gfCNCPoint5[25189] = {X 489.1455, Y 22.6360, Z -7.1667, A 0.000, B 0.000, C 0.000 }
gfCNCPoint5[25190] = {X 493.1303, Y 22.2874, Z -7.1667, A 0.000, B 0.000, C 0.000 }
gfCNCPoint5[25191] = {X 485.1607, Y 22.3674, Z -7.1667, A 0.000, B 0.000, C 0.000 }
gfCNCPoint5[25192] = {X 489.1455, Y 22.7160, Z -7.1667, A 0.000, B 0.000, C 0.000 }
gfCNCPoint5[25193] = {X 493.5290, Y 22.7160, Z -7.1667, A 0.000, B 0.000, C 0.000 }
gfCNCPoint5[25194] = {X 493.5290, Y 19.6226, Z -7.1667, A 0.000, B 0.000, C 0.000 }
gfCNCPoint5[25195] = {X 487.6640, Y 19.6221, Z -7.1667, A 0.000, B 0.000, C 0.000 }
gfCNCPoint5[25196] = {X 486.9712, Y 19.6268, Z -7.1667, A 0.000, B 0.000, C 0.000 }
gfCNCPoint5[25197] = {X 485.8542, Y 19.6990, Z -7.1667, A 0.000, B 0.000, C 0.000 }
gfCNCPoint5[25198] = {X 484.7569, Y 19.9204, Z -7.1667, A 0.000, B 0.000, C 0.000 }
gfCNCPoint5[25199] = {X 484.5580, Y 20.0321, Z -7.1667, A 0.000, B 0.000, C 0.000 }
gfCNCPoint5[25200] = {X 484.4352, Y 20.2245, Z -7.1667, A 0.000, B 0.000, C 0.000 }
gfCNCPoint5[25201] = {X 484.2684, Y 20.9674, Z -7.1667, A 0.000, B 0.000, C 0.000 }
gfCNCPoint5[25202] = {X 484.2552, Y 21.7288, Z -7.1667, A 0.000, B 0.000, C 0.000 }
gfCNCPoint5[25203] = {X 484.3961, Y 22.4771, Z -7.1667, A 0.000, B 0.000, C 0.000 }
gfCNCPoint5[25204] = {X 484.6514, Y 22.5532, Z -7.1667, A 0.000, B 0.000, C 0.000 }
gfCNCPoint5[25205] = {X 484.9147, Y 22.5933, Z -7.1667, A 0.000, B 0.000, C 0.000 }
gfCNCPoint5[25206] = {X 486.2771, Y 22.6950, Z -7.1667, A 0.000, B 0.000, C 0.000 }
gfCNCPoint5[25207] = {X 487.6431, Y 22.7160, Z -7.1667, A 0.000, B 0.000, C 0.000 }
gfCNCPoint5[25208] = {X 489.1455, Y 22.7160, Z -7.1667, A 0.000, B 0.000, C 0.000 }
gfCNCPoint5[25209] = {X 493.1303, Y 22.3674, Z -7.1667, A 0.000, B 0.000, C 0.000 }
gfCNCPoint5[25210] = {X 485.1607, Y 22.4474, Z -7.1667, A 0.000, B 0.000, C 0.000 }
gfCNCPoint5[25211] = {X 489.1455, Y 22.7960, Z -7.1667, A 0.000, B 0.000, C 0.000 }
gfCNCPoint5[25212] = {X 493.6090, Y 22.7960, Z -7.1667, A 0.000, B 0.000, C 0.000 }
gfCNCPoint5[25213] = {X 493.6090, Y 19.5426, Z -7.1667, A 0.000, B 0.000, C 0.000 }
gfCNCPoint5[25214] = {X 487.6637, Y 19.5421, Z -7.1667, A 0.000, B 0.000, C 0.000 }
gfCNCPoint5[25215] = {X 486.9710, Y 19.5468, Z -7.1667, A 0.000, B 0.000, C 0.000 }
gfCNCPoint5[25216] = {X 485.8434, Y 19.6197, Z -7.1667, A 0.000, B 0.000, C 0.000 }
gfCNCPoint5[25217] = {X 484.7359, Y 19.8432, Z -7.1667, A 0.000, B 0.000, C 0.000 }
gfCNCPoint5[25218] = {X 484.5030, Y 19.9740, Z -7.1667, A 0.000, B 0.000, C 0.000 }
gfCNCPoint5[25219] = {X 484.3593, Y 20.1991, Z -7.1667, A 0.000, B 0.000, C 0.000 }
gfCNCPoint5[25220] = {X 484.1874, Y 20.9710, Z -7.1667, A 0.000, B 0.000, C 0.000 }
gfCNCPoint5[25221] = {X 484.1778, Y 21.7618, Z -7.1667, A 0.000, B 0.000, C 0.000 }
gfCNCPoint5[25222] = {X 484.3308, Y 22.5376, Z -7.1667, A 0.000, B 0.000, C 0.000 }
gfCNCPoint5[25223] = {X 484.6140, Y 22.6267, Z -7.1667, A 0.000, B 0.000, C 0.000 }
gfCNCPoint5[25224] = {X 484.9073, Y 22.6730, Z -7.1667, A 0.000, B 0.000, C 0.000 }
gfCNCPoint5[25225] = {X 486.2736, Y 22.7749, Z -7.1667, A 0.000, B 0.000, C 0.000 }
gfCNCPoint5[25226] = {X 487.6437, Y 22.7960, Z -7.1667, A 0.000, B 0.000, C 0.000 }
gfCNCPoint5[25227] = {X 489.1455, Y 22.7960, Z -7.1667, A 0.000, B 0.000, C 0.000 }
gfCNCPoint5[25228] = {X 493.1303, Y 22.4474, Z -7.1667, A 0.000, B 0.000, C 0.000 }
gfCNCPoint5[25229] = {X 485.1607, Y 22.5274, Z -7.1667, A 0.000, B 0.000, C 0.000 }
gfCNCPoint5[25230] = {X 489.1455, Y 22.8760, Z -7.1667, A 0.000, B 0.000, C 0.000 }
gfCNCPoint5[25231] = {X 493.6890, Y 22.8760, Z -7.1667, A 0.000, B 0.000, C 0.000 }
gfCNCPoint5[25232] = {X 493.6890, Y 19.4626, Z -7.1667, A 0.000, B 0.000, C 0.000 }
gfCNCPoint5[25233] = {X 487.6634, Y 19.4621, Z -7.1667, A 0.000, B 0.000, C 0.000 }
gfCNCPoint5[25234] = {X 486.9708, Y 19.4668, Z -7.1667, A 0.000, B 0.000, C 0.000 }
gfCNCPoint5[25235] = {X 485.8327, Y 19.5404, Z -7.1667, A 0.000, B 0.000, C 0.000 }
gfCNCPoint5[25236] = {X 484.7148, Y 19.7660, Z -7.1667, A 0.000, B 0.000, C 0.000 }
gfCNCPoint5[25237] = {X 484.4481, Y 19.9159, Z -7.1667, A 0.000, B 0.000, C 0.000 }
gfCNCPoint5[25238] = {X 484.2835, Y 20.1737, Z -7.1667, A 0.000, B 0.000, C 0.000 }
gfCNCPoint5[25239] = {X 484.1065, Y 20.9744, Z -7.1667, A 0.000, B 0.000, C 0.000 }
gfCNCPoint5[25240] = {X 484.1005, Y 21.7943, Z -7.1667, A 0.000, B 0.000, C 0.000 }
gfCNCPoint5[25241] = {X 484.2657, Y 22.5974, Z -7.1667, A 0.000, B 0.000, C 0.000 }
gfCNCPoint5[25242] = {X 484.5771, Y 22.7001, Z -7.1667, A 0.000, B 0.000, C 0.000 }
gfCNCPoint5[25243] = {X 484.9007, Y 22.7527, Z -7.1667, A 0.000, B 0.000, C 0.000 }
gfCNCPoint5[25244] = {X 486.2706, Y 22.8548, Z -7.1667, A 0.000, B 0.000, C 0.000 }
gfCNCPoint5[25245] = {X 487.6442, Y 22.8760, Z -7.1667, A 0.000, B 0.000, C 0.000 }
gfCNCPoint5[25246] = {X 489.1455, Y 22.8760, Z -7.1667, A 0.000, B 0.000, C 0.000 }
gfCNCPoint5[25247] = {X 493.1303, Y 22.5274, Z -7.1667, A 0.000, B 0.000, C 0.000 }
gfCNCPoint5[25248] = {X 489.1455, Y 20.9560, Z -7.1667, A 0.000, B 0.000, C 0.000 }
gfCNCPoint5[25249] = {X 489.1455, Y 22.9560, Z -7.1667, A 0.000, B 0.000, C 0.000 }
gfCNCPoint5[25250] = {X 493.7690, Y 22.9560, Z -7.1667, A 0.000, B 0.000, C 0.000 }
gfCNCPoint5[25251] = {X 493.7690, Y 19.3826, Z -7.1667, A 0.000, B 0.000, C 0.000 }
gfCNCPoint5[25252] = {X 487.6632, Y 19.3821, Z -7.1667, A 0.000, B 0.000, C 0.000 }
gfCNCPoint5[25253] = {X 486.9707, Y 19.3868, Z -7.1667, A 0.000, B 0.000, C 0.000 }
gfCNCPoint5[25254] = {X 485.8220, Y 19.4611, Z -7.1667, A 0.000, B 0.000, C 0.000 }
gfCNCPoint5[25255] = {X 484.6937, Y 19.6888, Z -7.1667, A 0.000, B 0.000, C 0.000 }
gfCNCPoint5[25256] = {X 484.3931, Y 19.8577, Z -7.1667, A 0.000, B 0.000, C 0.000 }
gfCNCPoint5[25257] = {X 484.2076, Y 20.1484, Z -7.1667, A 0.000, B 0.000, C 0.000 }
gfCNCPoint5[25258] = {X 484.0256, Y 20.9775, Z -7.1667, A 0.000, B 0.000, C 0.000 }
gfCNCPoint5[25259] = {X 484.0233, Y 21.8264, Z -7.1667, A 0.000, B 0.000, C 0.000 }
gfCNCPoint5[25260] = {X 484.2007, Y 22.6566, Z -7.1667, A 0.000, B 0.000, C 0.000 }
gfCNCPoint5[25261] = {X 484.5397, Y 22.7732, Z -7.1667, A 0.000, B 0.000, C 0.000 }
gfCNCPoint5[25262] = {X 484.8932, Y 22.8324, Z -7.1667, A 0.000, B 0.000, C 0.000 }
gfCNCPoint5[25263] = {X 486.2672, Y 22.9348, Z -7.1667, A 0.000, B 0.000, C 0.000 }
gfCNCPoint5[25264] = {X 487.6448, Y 22.9560, Z -7.1667, A 0.000, B 0.000, C 0.000 }
gfCNCPoint5[25265] = {X 489.1455, Y 22.9560, Z -7.1667, A 0.000, B 0.000, C 0.000 }
gfCNCPoint5[25266] = {X 493.1455, Y 22.9560, Z -7.1667, A 0.000, B 0.000, C 0.000 }
gfCNCPoint5[25267] = {X 493.1455, Y 22.9560, Z -4.1667, A 0.000, B 0.000, C 0.000 }
gfCNCPoint5[25268] = {X 493.1455, Y 22.9560, Z 11.0000, A 0.000, B 0.000, C 0.000 }
gfCNCPoint5[25269] = {X 607.6967, Y 2.1241, Z 11.0000, A 0.000, B 0.000, C 0.000 }
gfCNCPoint5[25270] = {X 607.6967, Y 2.1241, Z -4.1667, A 0.000, B 0.000, C 0.000 }
gfCNCPoint5[25271] = {X 607.6967, Y 2.1241, Z -7.1667, A 0.000, B 0.000, C 0.000 }
gfCNCPoint5[25272] = {X 603.6967, Y 8.3204, Z -7.1667, A 0.000, B 0.000, C 0.000 }
gfCNCPoint5[25273] = {X 603.3211, Y 8.8203, Z -7.1667, A 0.000, B 0.000, C 0.000 }
gfCNCPoint5[25274] = {X 602.8784, Y 9.2620, Z -7.1667, A 0.000, B 0.000, C 0.000 }
gfCNCPoint5[25275] = {X 602.8782, Y 40.7378, Z -7.1667, A 0.000, B 0.000, C 0.000 }
gfCNCPoint5[25276] = {X 603.3210, Y 41.1795, Z -7.1667, A 0.000, B 0.000, C 0.000 }
gfCNCPoint5[25277] = {X 603.6967, Y 41.6796, Z -7.1667, A 0.000, B 0.000, C 0.000 }
gfCNCPoint5[25278] = {X 607.6967, Y 47.8759, Z -7.1667, A 0.000, B 0.000, C 0.000 }
gfCNCPoint5[25279] = {X 607.6967, Y 47.8759, Z -4.1667, A 0.000, B 0.000, C 0.000 }
gfCNCPoint5[25280] = {X 607.6967, Y 47.8759, Z 11.0000, A 0.000, B 0.000, C 0.000 }
gfCNCPoint5[25281] = {X 607.6967, Y 1.5441, Z 11.0000, A 0.000, B 0.000, C 0.000 }
gfCNCPoint5[25282] = {X 607.6967, Y 1.5441, Z -4.1667, A 0.000, B 0.000, C 0.000 }
gfCNCPoint5[25283] = {X 607.6967, Y 1.5441, Z -7.1667, A 0.000, B 0.000, C 0.000 }
gfCNCPoint5[25284] = {X 603.6967, Y 8.1709, Z -7.1667, A 0.000, B 0.000, C 0.000 }
gfCNCPoint5[25285] = {X 603.2902, Y 8.7357, Z -7.1667, A 0.000, B 0.000, C 0.000 }
gfCNCPoint5[25286] = {X 602.7984, Y 9.2280, Z -7.1667, A 0.000, B 0.000, C 0.000 }
gfCNCPoint5[25287] = {X 602.7982, Y 40.7725, Z -7.1667, A 0.000, B 0.000, C 0.000 }
gfCNCPoint5[25288] = {X 603.2901, Y 41.2647, Z -7.1667, A 0.000, B 0.000, C 0.000 }
gfCNCPoint5[25289] = {X 603.6967, Y 41.8295, Z -7.1667, A 0.000, B 0.000, C 0.000 }
gfCNCPoint5[25290] = {X 607.6967, Y 48.4531, Z -7.1667, A 0.000, B 0.000, C 0.000 }
gfCNCPoint5[25291] = {X 607.6967, Y 48.4531, Z -4.1667, A 0.000, B 0.000, C 0.000 }
gfCNCPoint5[25292] = {X 607.6967, Y 48.4531, Z 11.0000, A 0.000, B 0.000, C 0.000 }
gfCNCPoint5[25293] = {X 607.6967, Y 0.8767, Z 11.0000, A 0.000, B 0.000, C 0.000 }
gfCNCPoint5[25294] = {X 607.6967, Y 0.8767, Z -4.1667, A 0.000, B 0.000, C 0.000 }
gfCNCPoint5[25295] = {X 607.6967, Y 0.8767, Z -7.1667, A 0.000, B 0.000, C 0.000 }
gfCNCPoint5[25296] = {X 603.6967, Y 8.0118, Z -7.1667, A 0.000, B 0.000, C 0.000 }
gfCNCPoint5[25297] = {X 603.2612, Y 8.6459, Z -7.1667, A 0.000, B 0.000, C 0.000 }
gfCNCPoint5[25298] = {X 602.7184, Y 9.1908, Z -7.1667, A 0.000, B 0.000, C 0.000 }
gfCNCPoint5[25299] = {X 602.7182, Y 40.8097, Z -7.1667, A 0.000, B 0.000, C 0.000 }
gfCNCPoint5[25300] = {X 603.2611, Y 41.3545, Z -7.1667, A 0.000, B 0.000, C 0.000 }
gfCNCPoint5[25301] = {X 603.6967, Y 41.9885, Z -7.1667, A 0.000, B 0.000, C 0.000 }
gfCNCPoint5[25302] = {X 607.6967, Y 49.1198, Z -7.1667, A 0.000, B 0.000, C 0.000 }
gfCNCPoint5[25303] = {X 607.6967, Y 49.1198, Z -4.1667, A 0.000, B 0.000, C 0.000 }
gfCNCPoint5[25304] = {X 607.6967, Y 49.1198, Z 11.0000, A 0.000, B 0.000, C 0.000 }
gfCNCPoint5[25305] = {X 607.6952, Y 0.0778, Z 11.0000, A 0.000, B 0.000, C 0.000 }
gfCNCPoint5[25306] = {X 607.6952, Y 0.0778, Z -4.1667, A 0.000, B 0.000, C 0.000 }
gfCNCPoint5[25307] = {X 607.6952, Y 0.0778, Z -7.1667, A 0.000, B 0.000, C 0.000 }
gfCNCPoint5[25308] = {X 603.6967, Y 7.8429, Z -7.1667, A 0.000, B 0.000, C 0.000 }
gfCNCPoint5[25309] = {X 603.2345, Y 8.5522, Z -7.1667, A 0.000, B 0.000, C 0.000 }
gfCNCPoint5[25310] = {X 602.6384, Y 9.1532, Z -7.1667, A 0.000, B 0.000, C 0.000 }
gfCNCPoint5[25311] = {X 602.6382, Y 40.8473, Z -7.1667, A 0.000, B 0.000, C 0.000 }
gfCNCPoint5[25312] = {X 603.2344, Y 41.4482, Z -7.1667, A 0.000, B 0.000, C 0.000 }
gfCNCPoint5[25313] = {X 603.6967, Y 42.1573, Z -7.1667, A 0.000, B 0.000, C 0.000 }
gfCNCPoint5[25314] = {X 607.6967, Y 49.9206, Z -7.1667, A 0.000, B 0.000, C 0.000 }
gfCNCPoint5[25315] = {X 607.6967, Y 49.9206, Z -4.1667, A 0.000, B 0.000, C 0.000 }
gfCNCPoint5[25316] = {X 607.6967, Y 49.9206, Z 11.0000, A 0.000, B 0.000, C 0.000 }
gfCNCPoint5[25317] = {X 607.6538, Y -0.8117, Z 11.0000, A 0.000, B 0.000, C 0.000 }
gfCNCPoint5[25318] = {X 607.6538, Y -0.8117, Z -4.1667, A 0.000, B 0.000, C 0.000 }
gfCNCPoint5[25319] = {X 607.6538, Y -0.8117, Z -7.1667, A 0.000, B 0.000, C 0.000 }
gfCNCPoint5[25320] = {X 603.6967, Y 7.6606, Z -7.1667, A 0.000, B 0.000, C 0.000 }
gfCNCPoint5[25321] = {X 603.2075, Y 8.4556, Z -7.1667, A 0.000, B 0.000, C 0.000 }
gfCNCPoint5[25322] = {X 602.5505, Y 9.1186, Z -7.1667, A 0.000, B 0.000, C 0.000 }
gfCNCPoint5[25323] = {X 602.5584, Y 9.1532, Z -7.1667, A 0.000, B 0.000, C 0.000 }
gfCNCPoint5[25324] = {X 602.5582, Y 40.8854, Z -7.1667, A 0.000, B 0.000, C 0.000 }
gfCNCPoint5[25325] = {X 603.2107, Y 41.5469, Z -7.1667, A 0.000, B 0.000, C 0.000 }
gfCNCPoint5[25326] = {X 603.6967, Y 42.3390, Z -7.1667, A 0.000, B 0.000, C 0.000 }
gfCNCPoint5[25327] = {X 607.6967, Y 50.9203, Z -7.1667, A 0.000, B 0.000, C 0.000 }
gfCNCPoint5[25328] = {X 607.6967, Y 50.9203, Z -4.1667, A 0.000, B 0.000, C 0.000 }
gfCNCPoint5[25329] = {X 607.6967, Y 50.9203, Z 11.0000, A 0.000, B 0.000, C 0.000 }
gfCNCPoint5[25330] = {X 607.4985, Y -1.7359, Z 11.0000, A 0.000, B 0.000, C 0.000 }
gfCNCPoint5[25331] = {X 607.4985, Y -1.7359, Z -4.1667, A 0.000, B 0.000, C 0.000 }
gfCNCPoint5[25332] = {X 607.4985, Y -1.7359, Z -7.1667, A 0.000, B 0.000, C 0.000 }
gfCNCPoint5[25333] = {X 603.6967, Y 7.4620, Z -7.1667, A 0.000, B 0.000, C 0.000 }
gfCNCPoint5[25334] = {X 603.3770, Y 8.0779, Z -7.1667, A 0.000, B 0.000, C 0.000 }
gfCNCPoint5[25335] = {X 602.9557, Y 8.6292, Z -7.1667, A 0.000, B 0.000, C 0.000 }
gfCNCPoint5[25336] = {X 602.4454, Y 9.0995, Z -7.1667, A 0.000, B 0.000, C 0.000 }
gfCNCPoint5[25337] = {X 602.4784, Y 9.1532, Z -7.1667, A 0.000, B 0.000, C 0.000 }
gfCNCPoint5[25338] = {X 602.4782, Y 40.9223, Z -7.1667, A 0.000, B 0.000, C 0.000 }
gfCNCPoint5[25339] = {X 602.5731, Y 41.0034, Z -7.1667, A 0.000, B 0.000, C 0.000 }
gfCNCPoint5[25340] = {X 603.2274, Y 41.7029, Z -7.1667, A 0.000, B 0.000, C 0.000 }
gfCNCPoint5[25341] = {X 603.6967, Y 42.5380, Z -7.1667, A 0.000, B 0.000, C 0.000 }
gfCNCPoint5[25342] = {X 607.6967, Y 52.2154, Z -7.1667, A 0.000, B 0.000, C 0.000 }
gfCNCPoint5[25343] = {X 607.6967, Y 52.2154, Z -4.1667, A 0.000, B 0.000, C 0.000 }
gfCNCPoint5[25344] = {X 607.6967, Y 52.2154, Z 11.0000, A 0.000, B 0.000, C 0.000 }
gfCNCPoint5[25345] = {X 607.6967, Y 2.1238, Z 11.0000, A 0.000, B 0.000, C 0.000 }
gfCNCPoint5[25346] = {X 607.6967, Y 2.1238, Z -5.0000, A 0.000, B 0.000, C 0.000 }
gfCNCPoint5[25347] = {X 607.6967, Y 2.1238, Z -8.0000, A 0.000, B 0.000, C 0.000 }
gfCNCPoint5[25348] = {X 603.6967, Y 8.3204, Z -8.0000, A 0.000, B 0.000, C 0.000 }
gfCNCPoint5[25349] = {X 603.3212, Y 8.8202, Z -8.0000, A 0.000, B 0.000, C 0.000 }
gfCNCPoint5[25350] = {X 602.8787, Y 9.2617, Z -8.0000, A 0.000, B 0.000, C 0.000 }
gfCNCPoint5[25351] = {X 602.8785, Y 40.7381, Z -8.0000, A 0.000, B 0.000, C 0.000 }
gfCNCPoint5[25352] = {X 603.3211, Y 41.1797, Z -8.0000, A 0.000, B 0.000, C 0.000 }
gfCNCPoint5[25353] = {X 603.6967, Y 41.6796, Z -8.0000, A 0.000, B 0.000, C 0.000 }
gfCNCPoint5[25354] = {X 607.6967, Y 47.8762, Z -8.0000, A 0.000, B 0.000, C 0.000 }
gfCNCPoint5[25355] = {X 607.6967, Y 47.8762, Z -5.0000, A 0.000, B 0.000, C 0.000 }
gfCNCPoint5[25356] = {X 607.6967, Y 47.8762, Z 11.0000, A 0.000, B 0.000, C 0.000 }
gfCNCPoint5[25357] = {X 607.6967, Y 1.5428, Z 11.0000, A 0.000, B 0.000, C 0.000 }
gfCNCPoint5[25358] = {X 607.6967, Y 1.5428, Z -5.0000, A 0.000, B 0.000, C 0.000 }
gfCNCPoint5[25359] = {X 607.6967, Y 1.5428, Z -8.0000, A 0.000, B 0.000, C 0.000 }
gfCNCPoint5[25360] = {X 603.6967, Y 8.1709, Z -8.0000, A 0.000, B 0.000, C 0.000 }
gfCNCPoint5[25361] = {X 603.2904, Y 8.7357, Z -8.0000, A 0.000, B 0.000, C 0.000 }
gfCNCPoint5[25362] = {X 602.7987, Y 9.2280, Z -8.0000, A 0.000, B 0.000, C 0.000 }
gfCNCPoint5[25363] = {X 602.7985, Y 40.7725, Z -8.0000, A 0.000, B 0.000, C 0.000 }
gfCNCPoint5[25364] = {X 603.2903, Y 41.2647, Z -8.0000, A 0.000, B 0.000, C 0.000 }
gfCNCPoint5[25365] = {X 603.6967, Y 41.8294, Z -8.0000, A 0.000, B 0.000, C 0.000 }
gfCNCPoint5[25366] = {X 607.6967, Y 48.4543, Z -8.0000, A 0.000, B 0.000, C 0.000 }
gfCNCPoint5[25367] = {X 607.6967, Y 48.4543, Z -5.0000, A 0.000, B 0.000, C 0.000 }
gfCNCPoint5[25368] = {X 607.6967, Y 48.4543, Z 11.0000, A 0.000, B 0.000, C 0.000 }
gfCNCPoint5[25369] = {X 607.6967, Y 0.8752, Z 11.0000, A 0.000, B 0.000, C 0.000 }
gfCNCPoint5[25370] = {X 607.6967, Y 0.8752, Z -5.0000, A 0.000, B 0.000, C 0.000 }
gfCNCPoint5[25371] = {X 607.6967, Y 0.8752, Z -8.0000, A 0.000, B 0.000, C 0.000 }
gfCNCPoint5[25372] = {X 603.6967, Y 8.0119, Z -8.0000, A 0.000, B 0.000, C 0.000 }
gfCNCPoint5[25373] = {X 603.2614, Y 8.6459, Z -8.0000, A 0.000, B 0.000, C 0.000 }
gfCNCPoint5[25374] = {X 602.7187, Y 9.1908, Z -8.0000, A 0.000, B 0.000, C 0.000 }
gfCNCPoint5[25375] = {X 602.7185, Y 40.8097, Z -8.0000, A 0.000, B 0.000, C 0.000 }
gfCNCPoint5[25376] = {X 603.2612, Y 41.3545, Z -8.0000, A 0.000, B 0.000, C 0.000 }
gfCNCPoint5[25377] = {X 603.6967, Y 41.9884, Z -8.0000, A 0.000, B 0.000, C 0.000 }
gfCNCPoint5[25378] = {X 607.6967, Y 49.1213, Z -8.0000, A 0.000, B 0.000, C 0.000 }
gfCNCPoint5[25379] = {X 607.6967, Y 49.1213, Z -5.0000, A 0.000, B 0.000, C 0.000 }
gfCNCPoint5[25380] = {X 607.6967, Y 49.1213, Z 11.0000, A 0.000, B 0.000, C 0.000 }
gfCNCPoint5[25381] = {X 607.6952, Y 0.0758, Z 11.0000, A 0.000, B 0.000, C 0.000 }
gfCNCPoint5[25382] = {X 607.6952, Y 0.0758, Z -5.0000, A 0.000, B 0.000, C 0.000 }
gfCNCPoint5[25383] = {X 607.6952, Y 0.0758, Z -8.0000, A 0.000, B 0.000, C 0.000 }
gfCNCPoint5[25384] = {X 603.6967, Y 7.8429, Z -8.0000, A 0.000, B 0.000, C 0.000 }
gfCNCPoint5[25385] = {X 603.2347, Y 8.5522, Z -8.0000, A 0.000, B 0.000, C 0.000 }
gfCNCPoint5[25386] = {X 602.6387, Y 9.1532, Z -8.0000, A 0.000, B 0.000, C 0.000 }
gfCNCPoint5[25387] = {X 602.6385, Y 40.8473, Z -8.0000, A 0.000, B 0.000, C 0.000 }
gfCNCPoint5[25388] = {X 603.2346, Y 41.4482, Z -8.0000, A 0.000, B 0.000, C 0.000 }
gfCNCPoint5[25389] = {X 603.6967, Y 42.1573, Z -8.0000, A 0.000, B 0.000, C 0.000 }
gfCNCPoint5[25390] = {X 607.6967, Y 49.9225, Z -8.0000, A 0.000, B 0.000, C 0.000 }
gfCNCPoint5[25391] = {X 607.6967, Y 49.9225, Z -5.0000, A 0.000, B 0.000, C 0.000 }
gfCNCPoint5[25392] = {X 607.6967, Y 49.9225, Z 11.0000, A 0.000, B 0.000, C 0.000 }
gfCNCPoint5[25393] = {X 607.6537, Y -0.8120, Z 11.0000, A 0.000, B 0.000, C 0.000 }
gfCNCPoint5[25394] = {X 607.6537, Y -0.8120, Z -5.0000, A 0.000, B 0.000, C 0.000 }
gfCNCPoint5[25395] = {X 607.6537, Y -0.8120, Z -8.0000, A 0.000, B 0.000, C 0.000 }
gfCNCPoint5[25396] = {X 603.6967, Y 7.6606, Z -8.0000, A 0.000, B 0.000, C 0.000 }
gfCNCPoint5[25397] = {X 603.2076, Y 8.4555, Z -8.0000, A 0.000, B 0.000, C 0.000 }
gfCNCPoint5[25398] = {X 602.5507, Y 9.1184, Z -8.0000, A 0.000, B 0.000, C 0.000 }
gfCNCPoint5[25399] = {X 602.5587, Y 9.1532, Z -8.0000, A 0.000, B 0.000, C 0.000 }
gfCNCPoint5[25400] = {X 602.5585, Y 40.8854, Z -8.0000, A 0.000, B 0.000, C 0.000 }
gfCNCPoint5[25401] = {X 603.2109, Y 41.5470, Z -8.0000, A 0.000, B 0.000, C 0.000 }
gfCNCPoint5[25402] = {X 603.6967, Y 42.3390, Z -8.0000, A 0.000, B 0.000, C 0.000 }
gfCNCPoint5[25403] = {X 607.6967, Y 50.9229, Z -8.0000, A 0.000, B 0.000, C 0.000 }
gfCNCPoint5[25404] = {X 607.6967, Y 50.9229, Z -5.0000, A 0.000, B 0.000, C 0.000 }
gfCNCPoint5[25405] = {X 607.6967, Y 50.9229, Z 11.0000, A 0.000, B 0.000, C 0.000 }
gfCNCPoint5[25406] = {X 607.4984, Y -1.7363, Z 11.0000, A 0.000, B 0.000, C 0.000 }
gfCNCPoint5[25407] = {X 607.4984, Y -1.7363, Z -5.0000, A 0.000, B 0.000, C 0.000 }
gfCNCPoint5[25408] = {X 607.4984, Y -1.7363, Z -8.0000, A 0.000, B 0.000, C 0.000 }
gfCNCPoint5[25409] = {X 603.6967, Y 7.4620, Z -8.0000, A 0.000, B 0.000, C 0.000 }
gfCNCPoint5[25410] = {X 603.3770, Y 8.0778, Z -8.0000, A 0.000, B 0.000, C 0.000 }
gfCNCPoint5[25411] = {X 602.9557, Y 8.6292, Z -8.0000, A 0.000, B 0.000, C 0.000 }
gfCNCPoint5[25412] = {X 602.4454, Y 9.0995, Z -8.0000, A 0.000, B 0.000, C 0.000 }
gfCNCPoint5[25413] = {X 602.4787, Y 9.1532, Z -8.0000, A 0.000, B 0.000, C 0.000 }
gfCNCPoint5[25414] = {X 602.4785, Y 40.9221, Z -8.0000, A 0.000, B 0.000, C 0.000 }
gfCNCPoint5[25415] = {X 602.5732, Y 41.0035, Z -8.0000, A 0.000, B 0.000, C 0.000 }
gfCNCPoint5[25416] = {X 603.2275, Y 41.7030, Z -8.0000, A 0.000, B 0.000, C 0.000 }
gfCNCPoint5[25417] = {X 603.6967, Y 42.5380, Z -8.0000, A 0.000, B 0.000, C 0.000 }
gfCNCPoint5[25418] = {X 607.6967, Y 52.2160, Z -8.0000, A 0.000, B 0.000, C 0.000 }
gfCNCPoint5[25419] = {X 607.6967, Y 52.2160, Z -5.0000, A 0.000, B 0.000, C 0.000 }
gfCNCPoint5[25420] = {X 607.6967, Y 52.2160, Z 11.0000, A 0.000, B 0.000, C 0.000 }
gfCNCPoint5[25421] = {X 491.9949, Y 19.7827, Z 11.0000, A 0.000, B 0.000, C 0.000 }
gfCNCPoint5[25422] = {X 491.9949, Y 19.7827, Z -4.1667, A 0.000, B 0.000, C 0.000 }
gfCNCPoint5[25423] = {X 487.6645, Y 19.7824, Z -5.3270, A 0.000, B 0.000, C 0.000 }
gfCNCPoint5[25424] = {X 486.9696, Y 19.7871, Z -5.5132, A 0.000, B 0.000, C 0.000 }
gfCNCPoint5[25425] = {X 486.2694, Y 19.7852, Z -5.7008, A 0.000, B 0.000, C 0.000 }
gfCNCPoint5[25426] = {X 485.4747, Y 19.8906, Z -5.9156, A 0.000, B 0.000, C 0.000 }
gfCNCPoint5[25427] = {X 484.7992, Y 20.0750, Z -6.1032, A 0.000, B 0.000, C 0.000 }
gfCNCPoint5[25428] = {X 484.6645, Y 20.1118, Z -6.1407, A 0.000, B 0.000, C 0.000 }
gfCNCPoint5[25429] = {X 484.6309, Y 20.1437, Z -6.1531, A 0.000, B 0.000, C 0.000 }
gfCNCPoint5[25430] = {X 484.4396, Y 20.7178, Z -6.3152, A 0.000, B 0.000, C 0.000 }
gfCNCPoint5[25431] = {X 484.4058, Y 21.9039, Z -6.6332, A 0.000, B 0.000, C 0.000 }
gfCNCPoint5[25432] = {X 484.5275, Y 22.3532, Z -6.7579, A 0.000, B 0.000, C 0.000 }
gfCNCPoint5[25433] = {X 484.7223, Y 22.4164, Z -6.8128, A 0.000, B 0.000, C 0.000 }
gfCNCPoint5[25434] = {X 484.9347, Y 22.4342, Z -6.8699, A 0.000, B 0.000, C 0.000 }
gfCNCPoint5[25435] = {X 486.1049, Y 22.5561, Z -7.1851, A 0.000, B 0.000, C 0.000 }
gfCNCPoint5[25436] = {X 486.4629, Y 22.5722, Z -7.2812, A 0.000, B 0.000, C 0.000 }
gfCNCPoint5[25437] = {X 487.6448, Y 22.5560, Z -7.5979, A 0.000, B 0.000, C 0.000 }
gfCNCPoint5[25438] = {X 489.1455, Y 22.5560, Z -8.0000, A 0.000, B 0.000, C 0.000 }
gfCNCPoint5[25439] = {X 493.3690, Y 22.5560, Z -8.0000, A 0.000, B 0.000, C 0.000 }
gfCNCPoint5[25440] = {X 493.3690, Y 19.7828, Z -8.0000, A 0.000, B 0.000, C 0.000 }
gfCNCPoint5[25441] = {X 487.6645, Y 19.7824, Z -8.0000, A 0.000, B 0.000, C 0.000 }
gfCNCPoint5[25442] = {X 486.9696, Y 19.7871, Z -8.0000, A 0.000, B 0.000, C 0.000 }
gfCNCPoint5[25443] = {X 485.8747, Y 19.8579, Z -8.0000, A 0.000, B 0.000, C 0.000 }
gfCNCPoint5[25444] = {X 484.7992, Y 20.0750, Z -8.0000, A 0.000, B 0.000, C 0.000 }
gfCNCPoint5[25445] = {X 484.6678, Y 20.1489, Z -8.0000, A 0.000, B 0.000, C 0.000 }
gfCNCPoint5[25446] = {X 484.5867, Y 20.2762, Z -8.0000, A 0.000, B 0.000, C 0.000 }
gfCNCPoint5[25447] = {X 484.4310, Y 20.9602, Z -8.0000, A 0.000, B 0.000, C 0.000 }
gfCNCPoint5[25448] = {X 484.4110, Y 21.6614, Z -8.0000, A 0.000, B 0.000, C 0.000 }
gfCNCPoint5[25449] = {X 484.5275, Y 22.3532, Z -8.0000, A 0.000, B 0.000, C 0.000 }
gfCNCPoint5[25450] = {X 484.7287, Y 22.4057, Z -8.0000, A 0.000, B 0.000, C 0.000 }
gfCNCPoint5[25451] = {X 484.9347, Y 22.4342, Z -8.0000, A 0.000, B 0.000, C 0.000 }
gfCNCPoint5[25452] = {X 486.2879, Y 22.5350, Z -8.0000, A 0.000, B 0.000, C 0.000 }
gfCNCPoint5[25453] = {X 487.6448, Y 22.5560, Z -8.0000, A 0.000, B 0.000, C 0.000 }
gfCNCPoint5[25454] = {X 489.1455, Y 22.5560, Z -8.0000, A 0.000, B 0.000, C 0.000 }
gfCNCPoint5[25455] = {X 485.1607, Y 22.2874, Z -8.0000, A 0.000, B 0.000, C 0.000 }
gfCNCPoint5[25456] = {X 489.1455, Y 22.6360, Z -8.0000, A 0.000, B 0.000, C 0.000 }
gfCNCPoint5[25457] = {X 493.4490, Y 22.6360, Z -8.0000, A 0.000, B 0.000, C 0.000 }
gfCNCPoint5[25458] = {X 493.4490, Y 19.7028, Z -8.0000, A 0.000, B 0.000, C 0.000 }
gfCNCPoint5[25459] = {X 487.6642, Y 19.7024, Z -8.0000, A 0.000, B 0.000, C 0.000 }
gfCNCPoint5[25460] = {X 486.9713, Y 19.7072, Z -8.0000, A 0.000, B 0.000, C 0.000 }
gfCNCPoint5[25461] = {X 485.8649, Y 19.7785, Z -8.0000, A 0.000, B 0.000, C 0.000 }
gfCNCPoint5[25462] = {X 484.7782, Y 19.9979, Z -8.0000, A 0.000, B 0.000, C 0.000 }
gfCNCPoint5[25463] = {X 484.6128, Y 20.0908, Z -8.0000, A 0.000, B 0.000, C 0.000 }
gfCNCPoint5[25464] = {X 484.5108, Y 20.2509, Z -8.0000, A 0.000, B 0.000, C 0.000 }
gfCNCPoint5[25465] = {X 484.3498, Y 20.9643, Z -8.0000, A 0.000, B 0.000, C 0.000 }
gfCNCPoint5[25466] = {X 484.3333, Y 21.6955, Z -8.0000, A 0.000, B 0.000, C 0.000 }
gfCNCPoint5[25467] = {X 484.4617, Y 22.4155, Z -8.0000, A 0.000, B 0.000, C 0.000 }
gfCNCPoint5[25468] = {X 484.6884, Y 22.4790, Z -8.0000, A 0.000, B 0.000, C 0.000 }
gfCNCPoint5[25469] = {X 484.9212, Y 22.5133, Z -8.0000, A 0.000, B 0.000, C 0.000 }
gfCNCPoint5[25470] = {X 486.2801, Y 22.6147, Z -8.0000, A 0.000, B 0.000, C 0.000 }
gfCNCPoint5[25471] = {X 487.6426, Y 22.6360, Z -8.0000, A 0.000, B 0.000, C 0.000 }
gfCNCPoint5[25472] = {X 489.1455, Y 22.6360, Z -8.0000, A 0.000, B 0.000, C 0.000 }
gfCNCPoint5[25473] = {X 493.1303, Y 22.2874, Z -8.0000, A 0.000, B 0.000, C 0.000 }
gfCNCPoint5[25474] = {X 485.1607, Y 22.3674, Z -8.0000, A 0.000, B 0.000, C 0.000 }
gfCNCPoint5[25475] = {X 489.1455, Y 22.7160, Z -8.0000, A 0.000, B 0.000, C 0.000 }
gfCNCPoint5[25476] = {X 493.5290, Y 22.7160, Z -8.0000, A 0.000, B 0.000, C 0.000 }
gfCNCPoint5[25477] = {X 493.5290, Y 19.6228, Z -8.0000, A 0.000, B 0.000, C 0.000 }
gfCNCPoint5[25478] = {X 487.6640, Y 19.6224, Z -8.0000, A 0.000, B 0.000, C 0.000 }
gfCNCPoint5[25479] = {X 486.9712, Y 19.6272, Z -8.0000, A 0.000, B 0.000, C 0.000 }
gfCNCPoint5[25480] = {X 485.8542, Y 19.6992, Z -8.0000, A 0.000, B 0.000, C 0.000 }
gfCNCPoint5[25481] = {X 484.7571, Y 19.9207, Z -8.0000, A 0.000, B 0.000, C 0.000 }
gfCNCPoint5[25482] = {X 484.5578, Y 20.0327, Z -8.0000, A 0.000, B 0.000, C 0.000 }
gfCNCPoint5[25483] = {X 484.4349, Y 20.2256, Z -8.0000, A 0.000, B 0.000, C 0.000 }
gfCNCPoint5[25484] = {X 484.2688, Y 20.9681, Z -8.0000, A 0.000, B 0.000, C 0.000 }
gfCNCPoint5[25485] = {X 484.2557, Y 21.7290, Z -8.0000, A 0.000, B 0.000, C 0.000 }
gfCNCPoint5[25486] = {X 484.3962, Y 22.4768, Z -8.0000, A 0.000, B 0.000, C 0.000 }
gfCNCPoint5[25487] = {X 484.6514, Y 22.5529, Z -8.0000, A 0.000, B 0.000, C 0.000 }
gfCNCPoint5[25488] = {X 484.9147, Y 22.5930, Z -8.0000, A 0.000, B 0.000, C 0.000 }
gfCNCPoint5[25489] = {X 486.2771, Y 22.6947, Z -8.0000, A 0.000, B 0.000, C 0.000 }
gfCNCPoint5[25490] = {X 487.6431, Y 22.7160, Z -8.0000, A 0.000, B 0.000, C 0.000 }
gfCNCPoint5[25491] = {X 489.1455, Y 22.7160, Z -8.0000, A 0.000, B 0.000, C 0.000 }
gfCNCPoint5[25492] = {X 493.1303, Y 22.3674, Z -8.0000, A 0.000, B 0.000, C 0.000 }
gfCNCPoint5[25493] = {X 485.1607, Y 22.4474, Z -8.0000, A 0.000, B 0.000, C 0.000 }
gfCNCPoint5[25494] = {X 489.1455, Y 22.7960, Z -8.0000, A 0.000, B 0.000, C 0.000 }
gfCNCPoint5[25495] = {X 493.6090, Y 22.7960, Z -8.0000, A 0.000, B 0.000, C 0.000 }
gfCNCPoint5[25496] = {X 493.6090, Y 19.5428, Z -8.0000, A 0.000, B 0.000, C 0.000 }
gfCNCPoint5[25497] = {X 487.6637, Y 19.5424, Z -8.0000, A 0.000, B 0.000, C 0.000 }
gfCNCPoint5[25498] = {X 486.9710, Y 19.5472, Z -8.0000, A 0.000, B 0.000, C 0.000 }
gfCNCPoint5[25499] = {X 485.8435, Y 19.6200, Z -8.0000, A 0.000, B 0.000, C 0.000 }
gfCNCPoint5[25500] = {X 484.7360, Y 19.8435, Z -8.0000, A 0.000, B 0.000, C 0.000 }
gfCNCPoint5[25501] = {X 484.5028, Y 19.9746, Z -8.0000, A 0.000, B 0.000, C 0.000 }
gfCNCPoint5[25502] = {X 484.3590, Y 20.2003, Z -8.0000, A 0.000, B 0.000, C 0.000 }
gfCNCPoint5[25503] = {X 484.1878, Y 20.9718, Z -8.0000, A 0.000, B 0.000, C 0.000 }
gfCNCPoint5[25504] = {X 484.1783, Y 21.7619, Z -8.0000, A 0.000, B 0.000, C 0.000 }
gfCNCPoint5[25505] = {X 484.3309, Y 22.5373, Z -8.0000, A 0.000, B 0.000, C 0.000 }
gfCNCPoint5[25506] = {X 484.6145, Y 22.6265, Z -8.0000, A 0.000, B 0.000, C 0.000 }
gfCNCPoint5[25507] = {X 484.9081, Y 22.6727, Z -8.0000, A 0.000, B 0.000, C 0.000 }
gfCNCPoint5[25508] = {X 486.2741, Y 22.7746, Z -8.0000, A 0.000, B 0.000, C 0.000 }
gfCNCPoint5[25509] = {X 487.6437, Y 22.7960, Z -8.0000, A 0.000, B 0.000, C 0.000 }
gfCNCPoint5[25510] = {X 489.1455, Y 22.7960, Z -8.0000, A 0.000, B 0.000, C 0.000 }
gfCNCPoint5[25511] = {X 493.1303, Y 22.4474, Z -8.0000, A 0.000, B 0.000, C 0.000 }
gfCNCPoint5[25512] = {X 485.1607, Y 22.5274, Z -8.0000, A 0.000, B 0.000, C 0.000 }
gfCNCPoint5[25513] = {X 489.1455, Y 22.8760, Z -8.0000, A 0.000, B 0.000, C 0.000 }
gfCNCPoint5[25514] = {X 493.6890, Y 22.8760, Z -8.0000, A 0.000, B 0.000, C 0.000 }
gfCNCPoint5[25515] = {X 493.6890, Y 19.4628, Z -8.0000, A 0.000, B 0.000, C 0.000 }
gfCNCPoint5[25516] = {X 487.6634, Y 19.4624, Z -8.0000, A 0.000, B 0.000, C 0.000 }
gfCNCPoint5[25517] = {X 486.9708, Y 19.4671, Z -8.0000, A 0.000, B 0.000, C 0.000 }
gfCNCPoint5[25518] = {X 485.8328, Y 19.5407, Z -8.0000, A 0.000, B 0.000, C 0.000 }
gfCNCPoint5[25519] = {X 484.7150, Y 19.7663, Z -8.0000, A 0.000, B 0.000, C 0.000 }
gfCNCPoint5[25520] = {X 484.4478, Y 19.9165, Z -8.0000, A 0.000, B 0.000, C 0.000 }
gfCNCPoint5[25521] = {X 484.2831, Y 20.1750, Z -8.0000, A 0.000, B 0.000, C 0.000 }
gfCNCPoint5[25522] = {X 484.1069, Y 20.9752, Z -8.0000, A 0.000, B 0.000, C 0.000 }
gfCNCPoint5[25523] = {X 484.1010, Y 21.7945, Z -8.0000, A 0.000, B 0.000, C 0.000 }
gfCNCPoint5[25524] = {X 484.2657, Y 22.5971, Z -8.0000, A 0.000, B 0.000, C 0.000 }
gfCNCPoint5[25525] = {X 484.5771, Y 22.6998, Z -8.0000, A 0.000, B 0.000, C 0.000 }
gfCNCPoint5[25526] = {X 484.9007, Y 22.7524, Z -8.0000, A 0.000, B 0.000, C 0.000 }
gfCNCPoint5[25527] = {X 486.2706, Y 22.8545, Z -8.0000, A 0.000, B 0.000, C 0.000 }
gfCNCPoint5[25528] = {X 487.6442, Y 22.8760, Z -8.0000, A 0.000, B 0.000, C 0.000 }
gfCNCPoint5[25529] = {X 489.1455, Y 22.8760, Z -8.0000, A 0.000, B 0.000, C 0.000 }
gfCNCPoint5[25530] = {X 493.1303, Y 22.5274, Z -8.0000, A 0.000, B 0.000, C 0.000 }
gfCNCPoint5[25531] = {X 485.1607, Y 22.6074, Z -8.0000, A 0.000, B 0.000, C 0.000 }
gfCNCPoint5[25532] = {X 489.1455, Y 22.9560, Z -8.0000, A 0.000, B 0.000, C 0.000 }
gfCNCPoint5[25533] = {X 493.7690, Y 22.9560, Z -8.0000, A 0.000, B 0.000, C 0.000 }
gfCNCPoint5[25534] = {X 493.7690, Y 19.3829, Z -8.0000, A 0.000, B 0.000, C 0.000 }
gfCNCPoint5[25535] = {X 487.6632, Y 19.3824, Z -8.0000, A 0.000, B 0.000, C 0.000 }
gfCNCPoint5[25536] = {X 486.9707, Y 19.3871, Z -8.0000, A 0.000, B 0.000, C 0.000 }
gfCNCPoint5[25537] = {X 485.8221, Y 19.4614, Z -8.0000, A 0.000, B 0.000, C 0.000 }
gfCNCPoint5[25538] = {X 484.6939, Y 19.6891, Z -8.0000, A 0.000, B 0.000, C 0.000 }
gfCNCPoint5[25539] = {X 484.3928, Y 19.8584, Z -8.0000, A 0.000, B 0.000, C 0.000 }
gfCNCPoint5[25540] = {X 484.2072, Y 20.1497, Z -8.0000, A 0.000, B 0.000, C 0.000 }
gfCNCPoint5[25541] = {X 484.0261, Y 20.9784, Z -8.0000, A 0.000, B 0.000, C 0.000 }
gfCNCPoint5[25542] = {X 484.0239, Y 21.8266, Z -8.0000, A 0.000, B 0.000, C 0.000 }
gfCNCPoint5[25543] = {X 484.2007, Y 22.6562, Z -8.0000, A 0.000, B 0.000, C 0.000 }
gfCNCPoint5[25544] = {X 484.5397, Y 22.7729, Z -8.0000, A 0.000, B 0.000, C 0.000 }
gfCNCPoint5[25545] = {X 484.8932, Y 22.8320, Z -8.0000, A 0.000, B 0.000, C 0.000 }
gfCNCPoint5[25546] = {X 486.2672, Y 22.9345, Z -8.0000, A 0.000, B 0.000, C 0.000 }
gfCNCPoint5[25547] = {X 487.6448, Y 22.9560, Z -8.0000, A 0.000, B 0.000, C 0.000 }
gfCNCPoint5[25548] = {X 489.1455, Y 22.9560, Z -8.0000, A 0.000, B 0.000, C 0.000 }
gfCNCPoint5[25549] = {X 493.1303, Y 22.6074, Z -8.0000, A 0.000, B 0.000, C 0.000 }
gfCNCPoint5[25550] = {X 493.1303, Y 22.6074, Z -5.0000, A 0.000, B 0.000, C 0.000 }
gfCNCPoint5[25551] = {X 493.1303, Y 22.6074, Z 11.0000, A 0.000, B 0.000, C 0.000 }
gfCNCPoint5[25552] = {X 448.7159, Y 19.7829, Z 11.0000, A 0.000, B 0.000, C 0.000 }
gfCNCPoint5[25553] = {X 448.7159, Y 19.7829, Z -4.1667, A 0.000, B 0.000, C 0.000 }
gfCNCPoint5[25554] = {X 444.0414, Y 19.7831, Z -5.4192, A 0.000, B 0.000, C 0.000 }
gfCNCPoint5[25555] = {X 443.3486, Y 19.7993, Z -5.6049, A 0.000, B 0.000, C 0.000 }
gfCNCPoint5[25556] = {X 442.7492, Y 19.8059, Z -5.7655, A 0.000, B 0.000, C 0.000 }
gfCNCPoint5[25557] = {X 442.0371, Y 19.9292, Z -5.9591, A 0.000, B 0.000, C 0.000 }
gfCNCPoint5[25558] = {X 441.4703, Y 20.1243, Z -6.1198, A 0.000, B 0.000, C 0.000 }
gfCNCPoint5[25559] = {X 441.3675, Y 20.1597, Z -6.1489, A 0.000, B 0.000, C 0.000 }
gfCNCPoint5[25560] = {X 441.1899, Y 20.7194, Z -6.3062, A 0.000, B 0.000, C 0.000 }
gfCNCPoint5[25561] = {X 441.1563, Y 21.8870, Z -6.6192, A 0.000, B 0.000, C 0.000 }
gfCNCPoint5[25562] = {X 441.2744, Y 22.3506, Z -6.7474, A 0.000, B 0.000, C 0.000 }
gfCNCPoint5[25563] = {X 441.5051, Y 22.4259, Z -6.8124, A 0.000, B 0.000, C 0.000 }
gfCNCPoint5[25564] = {X 441.7467, Y 22.4476, Z -6.8774, A 0.000, B 0.000, C 0.000 }
gfCNCPoint5[25565] = {X 443.0211, Y 22.5620, Z -7.2203, A 0.000, B 0.000, C 0.000 }
gfCNCPoint5[25566] = {X 443.1117, Y 22.5657, Z -7.2446, A 0.000, B 0.000, C 0.000 }
gfCNCPoint5[25567] = {X 444.3942, Y 22.5560, Z -7.5882, A 0.000, B 0.000, C 0.000 }
gfCNCPoint5[25568] = {X 445.9310, Y 22.5560, Z -8.0000, A 0.000, B 0.000, C 0.000 }
gfCNCPoint5[25569] = {X 450.1184, Y 22.5560, Z -8.0000, A 0.000, B 0.000, C 0.000 }
gfCNCPoint5[25570] = {X 450.1184, Y 19.7829, Z -8.0000, A 0.000, B 0.000, C 0.000 }
gfCNCPoint5[25571] = {X 444.0414, Y 19.7831, Z -8.0000, A 0.000, B 0.000, C 0.000 }
gfCNCPoint5[25572] = {X 443.3486, Y 19.7993, Z -8.0000, A 0.000, B 0.000, C 0.000 }
gfCNCPoint5[25573] = {X 442.3964, Y 19.8864, Z -8.0000, A 0.000, B 0.000, C 0.000 }
gfCNCPoint5[25574] = {X 441.4703, Y 20.1243, Z -8.0000, A 0.000, B 0.000, C 0.000 }
gfCNCPoint5[25575] = {X 441.3860, Y 20.1777, Z -8.0000, A 0.000, B 0.000, C 0.000 }
gfCNCPoint5[25576] = {X 441.3346, Y 20.2634, Z -8.0000, A 0.000, B 0.000, C 0.000 }
gfCNCPoint5[25577] = {X 441.1848, Y 20.9514, Z -8.0000, A 0.000, B 0.000, C 0.000 }
gfCNCPoint5[25578] = {X 441.1645, Y 21.6551, Z -8.0000, A 0.000, B 0.000, C 0.000 }
gfCNCPoint5[25579] = {X 441.2744, Y 22.3506, Z -8.0000, A 0.000, B 0.000, C 0.000 }
gfCNCPoint5[25580] = {X 441.5078, Y 22.4125, Z -8.0000, A 0.000, B 0.000, C 0.000 }
gfCNCPoint5[25581] = {X 441.7467, Y 22.4476, Z -8.0000, A 0.000, B 0.000, C 0.000 }
gfCNCPoint5[25582] = {X 443.0692, Y 22.5340, Z -8.0000, A 0.000, B 0.000, C 0.000 }
gfCNCPoint5[25583] = {X 444.3942, Y 22.5560, Z -8.0000, A 0.000, B 0.000, C 0.000 }
gfCNCPoint5[25584] = {X 445.9310, Y 22.5560, Z -8.0000, A 0.000, B 0.000, C 0.000 }
gfCNCPoint5[25585] = {X 441.9462, Y 22.2874, Z -8.0000, A 0.000, B 0.000, C 0.000 }
gfCNCPoint5[25586] = {X 445.9310, Y 22.6360, Z -8.0000, A 0.000, B 0.000, C 0.000 }
gfCNCPoint5[25587] = {X 450.1984, Y 22.6360, Z -8.0000, A 0.000, B 0.000, C 0.000 }
gfCNCPoint5[25588] = {X 450.1984, Y 19.7029, Z -8.0000, A 0.000, B 0.000, C 0.000 }
gfCNCPoint5[25589] = {X 444.0404, Y 19.7031, Z -8.0000, A 0.000, B 0.000, C 0.000 }
gfCNCPoint5[25590] = {X 443.3497, Y 19.7193, Z -8.0000, A 0.000, B 0.000, C 0.000 }
gfCNCPoint5[25591] = {X 442.3838, Y 19.8074, Z -8.0000, A 0.000, B 0.000, C 0.000 }
gfCNCPoint5[25592] = {X 441.4443, Y 20.0486, Z -8.0000, A 0.000, B 0.000, C 0.000 }
gfCNCPoint5[25593] = {X 441.3287, Y 20.1219, Z -8.0000, A 0.000, B 0.000, C 0.000 }
gfCNCPoint5[25594] = {X 441.2583, Y 20.2392, Z -8.0000, A 0.000, B 0.000, C 0.000 }
gfCNCPoint5[25595] = {X 441.1036, Y 20.9561, Z -8.0000, A 0.000, B 0.000, C 0.000 }
gfCNCPoint5[25596] = {X 441.0866, Y 21.6893, Z -8.0000, A 0.000, B 0.000, C 0.000 }
gfCNCPoint5[25597] = {X 441.2079, Y 22.4125, Z -8.0000, A 0.000, B 0.000, C 0.000 }
gfCNCPoint5[25598] = {X 441.4702, Y 22.4863, Z -8.0000, A 0.000, B 0.000, C 0.000 }
gfCNCPoint5[25599] = {X 441.7396, Y 22.5273, Z -8.0000, A 0.000, B 0.000, C 0.000 }
gfCNCPoint5[25600] = {X 443.0650, Y 22.6139, Z -8.0000, A 0.000, B 0.000, C 0.000 }
gfCNCPoint5[25601] = {X 444.3930, Y 22.6360, Z -8.0000, A 0.000, B 0.000, C 0.000 }
gfCNCPoint5[25602] = {X 445.9310, Y 22.6360, Z -8.0000, A 0.000, B 0.000, C 0.000 }
gfCNCPoint5[25603] = {X 449.9157, Y 22.2874, Z -8.0000, A 0.000, B 0.000, C 0.000 }
gfCNCPoint5[25604] = {X 441.9462, Y 22.3674, Z -8.0000, A 0.000, B 0.000, C 0.000 }
gfCNCPoint5[25605] = {X 445.9310, Y 22.7160, Z -8.0000, A 0.000, B 0.000, C 0.000 }
gfCNCPoint5[25606] = {X 450.2784, Y 22.7160, Z -8.0000, A 0.000, B 0.000, C 0.000 }
gfCNCPoint5[25607] = {X 450.2784, Y 19.6229, Z -8.0000, A 0.000, B 0.000, C 0.000 }
gfCNCPoint5[25608] = {X 444.0395, Y 19.6231, Z -8.0000, A 0.000, B 0.000, C 0.000 }
gfCNCPoint5[25609] = {X 443.3483, Y 19.6393, Z -8.0000, A 0.000, B 0.000, C 0.000 }
gfCNCPoint5[25610] = {X 442.3699, Y 19.7286, Z -8.0000, A 0.000, B 0.000, C 0.000 }
gfCNCPoint5[25611] = {X 441.4183, Y 19.9730, Z -8.0000, A 0.000, B 0.000, C 0.000 }
gfCNCPoint5[25612] = {X 441.2714, Y 20.0660, Z -8.0000, A 0.000, B 0.000, C 0.000 }
gfCNCPoint5[25613] = {X 441.1821, Y 20.2150, Z -8.0000, A 0.000, B 0.000, C 0.000 }
gfCNCPoint5[25614] = {X 441.0226, Y 20.9606, Z -8.0000, A 0.000, B 0.000, C 0.000 }
gfCNCPoint5[25615] = {X 441.0089, Y 21.7229, Z -8.0000, A 0.000, B 0.000, C 0.000 }
gfCNCPoint5[25616] = {X 441.1417, Y 22.4737, Z -8.0000, A 0.000, B 0.000, C 0.000 }
gfCNCPoint5[25617] = {X 441.4327, Y 22.5599, Z -8.0000, A 0.000, B 0.000, C 0.000 }
gfCNCPoint5[25618] = {X 441.7325, Y 22.6070, Z -8.0000, A 0.000, B 0.000, C 0.000 }
gfCNCPoint5[25619] = {X 443.0616, Y 22.6938, Z -8.0000, A 0.000, B 0.000, C 0.000 }
gfCNCPoint5[25620] = {X 444.3933, Y 22.7160, Z -8.0000, A 0.000, B 0.000, C 0.000 }
gfCNCPoint5[25621] = {X 445.9310, Y 22.7160, Z -8.0000, A 0.000, B 0.000, C 0.000 }
gfCNCPoint5[25622] = {X 449.9157, Y 22.3674, Z -8.0000, A 0.000, B 0.000, C 0.000 }
gfCNCPoint5[25623] = {X 441.9462, Y 22.4474, Z -8.0000, A 0.000, B 0.000, C 0.000 }
gfCNCPoint5[25624] = {X 445.9310, Y 22.7960, Z -8.0000, A 0.000, B 0.000, C 0.000 }
gfCNCPoint5[25625] = {X 450.3584, Y 22.7960, Z -8.0000, A 0.000, B 0.000, C 0.000 }
gfCNCPoint5[25626] = {X 450.3584, Y 19.5429, Z -8.0000, A 0.000, B 0.000, C 0.000 }
gfCNCPoint5[25627] = {X 444.0385, Y 19.5431, Z -8.0000, A 0.000, B 0.000, C 0.000 }
gfCNCPoint5[25628] = {X 443.3469, Y 19.5593, Z -8.0000, A 0.000, B 0.000, C 0.000 }
gfCNCPoint5[25629] = {X 442.3560, Y 19.6498, Z -8.0000, A 0.000, B 0.000, C 0.000 }
gfCNCPoint5[25630] = {X 441.3922, Y 19.8974, Z -8.0000, A 0.000, B 0.000, C 0.000 }
gfCNCPoint5[25631] = {X 441.2142, Y 20.0101, Z -8.0000, A 0.000, B 0.000, C 0.000 }
gfCNCPoint5[25632] = {X 441.1058, Y 20.1908, Z -8.0000, A 0.000, B 0.000, C 0.000 }
gfCNCPoint5[25633] = {X 440.9416, Y 20.9649, Z -8.0000, A 0.000, B 0.000, C 0.000 }
gfCNCPoint5[25634] = {X 440.9314, Y 21.7562, Z -8.0000, A 0.000, B 0.000, C 0.000 }
gfCNCPoint5[25635] = {X 441.0757, Y 22.5342, Z -8.0000, A 0.000, B 0.000, C 0.000 }
gfCNCPoint5[25636] = {X 441.3951, Y 22.6334, Z -8.0000, A 0.000, B 0.000, C 0.000 }
gfCNCPoint5[25637] = {X 441.7253, Y 22.6867, Z -8.0000, A 0.000, B 0.000, C 0.000 }
gfCNCPoint5[25638] = {X 443.0582, Y 22.7738, Z -8.0000, A 0.000, B 0.000, C 0.000 }
gfCNCPoint5[25639] = {X 444.3936, Y 22.7960, Z -8.0000, A 0.000, B 0.000, C 0.000 }
gfCNCPoint5[25640] = {X 445.9310, Y 22.7960, Z -8.0000, A 0.000, B 0.000, C 0.000 }
gfCNCPoint5[25641] = {X 449.9157, Y 22.4474, Z -8.0000, A 0.000, B 0.000, C 0.000 }
gfCNCPoint5[25642] = {X 441.9462, Y 22.5274, Z -8.0000, A 0.000, B 0.000, C 0.000 }
gfCNCPoint5[25643] = {X 445.9310, Y 22.8760, Z -8.0000, A 0.000, B 0.000, C 0.000 }
gfCNCPoint5[25644] = {X 450.4384, Y 22.8760, Z -8.0000, A 0.000, B 0.000, C 0.000 }
gfCNCPoint5[25645] = {X 450.4384, Y 19.4629, Z -8.0000, A 0.000, B 0.000, C 0.000 }
gfCNCPoint5[25646] = {X 444.0376, Y 19.4631, Z -8.0000, A 0.000, B 0.000, C 0.000 }
gfCNCPoint5[25647] = {X 443.3456, Y 19.4793, Z -8.0000, A 0.000, B 0.000, C 0.000 }
gfCNCPoint5[25648] = {X 442.3421, Y 19.5710, Z -8.0000, A 0.000, B 0.000, C 0.000 }
gfCNCPoint5[25649] = {X 441.3662, Y 19.8217, Z -8.0000, A 0.000, B 0.000, C 0.000 }
gfCNCPoint5[25650] = {X 441.1569, Y 19.9542, Z -8.0000, A 0.000, B 0.000, C 0.000 }
gfCNCPoint5[25651] = {X 441.0296, Y 20.1666, Z -8.0000, A 0.000, B 0.000, C 0.000 }
gfCNCPoint5[25652] = {X 440.8606, Y 20.9691, Z -8.0000, A 0.000, B 0.000, C 0.000 }
gfCNCPoint5[25653] = {X 440.8540, Y 21.7891, Z -8.0000, A 0.000, B 0.000, C 0.000 }
gfCNCPoint5[25654] = {X 441.0099, Y 22.5941, Z -8.0000, A 0.000, B 0.000, C 0.000 }
gfCNCPoint5[25655] = {X 441.3576, Y 22.7067, Z -8.0000, A 0.000, B 0.000, C 0.000 }
gfCNCPoint5[25656] = {X 441.7182, Y 22.7664, Z -8.0000, A 0.000, B 0.000, C 0.000 }
gfCNCPoint5[25657] = {X 443.0547, Y 22.8537, Z -8.0000, A 0.000, B 0.000, C 0.000 }
gfCNCPoint5[25658] = {X 444.3939, Y 22.8760, Z -8.0000, A 0.000, B 0.000, C 0.000 }
gfCNCPoint5[25659] = {X 445.9310, Y 22.8760, Z -8.0000, A 0.000, B 0.000, C 0.000 }
gfCNCPoint5[25660] = {X 449.9157, Y 22.5274, Z -8.0000, A 0.000, B 0.000, C 0.000 }
gfCNCPoint5[25661] = {X 445.9310, Y 20.9560, Z -8.0000, A 0.000, B 0.000, C 0.000 }
gfCNCPoint5[25662] = {X 445.9310, Y 22.9560, Z -8.0000, A 0.000, B 0.000, C 0.000 }
gfCNCPoint5[25663] = {X 450.5184, Y 22.9560, Z -8.0000, A 0.000, B 0.000, C 0.000 }
gfCNCPoint5[25664] = {X 450.5184, Y 19.3829, Z -8.0000, A 0.000, B 0.000, C 0.000 }
gfCNCPoint5[25665] = {X 444.0367, Y 19.3831, Z -8.0000, A 0.000, B 0.000, C 0.000 }
gfCNCPoint5[25666] = {X 443.3442, Y 19.3993, Z -8.0000, A 0.000, B 0.000, C 0.000 }
gfCNCPoint5[25667] = {X 442.3282, Y 19.4922, Z -8.0000, A 0.000, B 0.000, C 0.000 }
gfCNCPoint5[25668] = {X 441.3401, Y 19.7461, Z -8.0000, A 0.000, B 0.000, C 0.000 }
gfCNCPoint5[25669] = {X 441.0997, Y 19.8984, Z -8.0000, A 0.000, B 0.000, C 0.000 }
gfCNCPoint5[25670] = {X 440.9533, Y 20.1425, Z -8.0000, A 0.000, B 0.000, C 0.000 }
gfCNCPoint5[25671] = {X 440.7798, Y 20.9731, Z -8.0000, A 0.000, B 0.000, C 0.000 }
gfCNCPoint5[25672] = {X 440.7767, Y 21.8216, Z -8.0000, A 0.000, B 0.000, C 0.000 }
gfCNCPoint5[25673] = {X 440.9444, Y 22.6535, Z -8.0000, A 0.000, B 0.000, C 0.000 }
gfCNCPoint5[25674] = {X 441.3201, Y 22.7798, Z -8.0000, A 0.000, B 0.000, C 0.000 }
gfCNCPoint5[25675] = {X 441.7110, Y 22.8460, Z -8.0000, A 0.000, B 0.000, C 0.000 }
gfCNCPoint5[25676] = {X 443.0513, Y 22.9336, Z -8.0000, A 0.000, B 0.000, C 0.000 }
gfCNCPoint5[25677] = {X 444.3942, Y 22.9560, Z -8.0000, A 0.000, B 0.000, C 0.000 }
gfCNCPoint5[25678] = {X 445.9310, Y 22.9560, Z -8.0000, A 0.000, B 0.000, C 0.000 }
gfCNCPoint5[25679] = {X 449.9310, Y 22.9560, Z -8.0000, A 0.000, B 0.000, C 0.000 }
gfCNCPoint5[25680] = {X 449.9310, Y 22.9560, Z -5.0000, A 0.000, B 0.000, C 0.000 }
gfCNCPoint5[25681] = {X 449.9310, Y 22.9560, Z 11.0000, A 0.000, B 0.000, C 0.000 }
gfCNCPoint5[25682] = {X 507.6811, Y 107.6952, Z 11.0000, A 0.000, B 0.000, C 0.000 }
gfCNCPoint5[25683] = {X 507.6811, Y 107.6952, Z -5.0000, A 0.000, B 0.000, C 0.000 }
gfCNCPoint5[25684] = {X 507.6811, Y 107.6952, Z -8.0000, A 0.000, B 0.000, C 0.000 }
gfCNCPoint5[25685] = {X 507.6811, Y 71.2952, Z -8.0000, A 0.000, B 0.000, C 0.000 }
gfCNCPoint5[25686] = {X 509.5505, Y 71.2952, Z -8.0000, A 0.000, B 0.000, C 0.000 }
gfCNCPoint5[25687] = {X 509.0280, Y 71.0692, Z -8.0000, A 0.000, B 0.000, C 0.000 }
gfCNCPoint5[25688] = {X 508.5105, Y 70.8320, Z -8.0000, A 0.000, B 0.000, C 0.000 }
gfCNCPoint5[25689] = {X 507.1671, Y 71.0985, Z -8.0000, A 0.000, B 0.000, C 0.000 }
gfCNCPoint5[25690] = {X 505.8117, Y 71.2952, Z -8.0000, A 0.000, B 0.000, C 0.000 }
gfCNCPoint5[25691] = {X 507.6811, Y 71.2952, Z -8.0000, A 0.000, B 0.000, C 0.000 }
gfCNCPoint5[25692] = {X 507.6811, Y 73.6952, Z -8.0000, A 0.000, B 0.000, C 0.000 }
gfCNCPoint5[25693] = {X 551.2538, Y 73.6952, Z -8.0000, A 0.000, B 0.000, C 0.000 }
gfCNCPoint5[25694] = {X 549.1246, Y 72.7709, Z -8.0000, A 0.000, B 0.000, C 0.000 }
gfCNCPoint5[25695] = {X 547.0710, Y 71.6890, Z -8.0000, A 0.000, B 0.000, C 0.000 }
gfCNCPoint5[25696] = {X 545.1047, Y 70.4554, Z -8.0000, A 0.000, B 0.000, C 0.000 }
gfCNCPoint5[25697] = {X 543.2369, Y 69.0773, Z -8.0000, A 0.000, B 0.000, C 0.000 }
gfCNCPoint5[25698] = {X 529.7624, Y 69.0775, Z -8.0000, A 0.000, B 0.000, C 0.000 }
gfCNCPoint5[25699] = {X 527.5519, Y 69.8798, Z -8.0000, A 0.000, B 0.000, C 0.000 }
gfCNCPoint5[25700] = {X 525.2740, Y 70.4641, Z -8.0000, A 0.000, B 0.000, C 0.000 }
gfCNCPoint5[25701] = {X 522.9502, Y 70.8249, Z -8.0000, A 0.000, B 0.000, C 0.000 }
gfCNCPoint5[25702] = {X 520.6023, Y 70.9588, Z -8.0000, A 0.000, B 0.000, C 0.000 }
gfCNCPoint5[25703] = {X 519.7998, Y 70.9591, Z -8.0000, A 0.000, B 0.000, C 0.000 }
gfCNCPoint5[25704] = {X 517.4111, Y 70.8404, Z -8.0000, A 0.000, B 0.000, C 0.000 }
gfCNCPoint5[25705] = {X 515.0461, Y 70.4852, Z -8.0000, A 0.000, B 0.000, C 0.000 }
gfCNCPoint5[25706] = {X 512.7279, Y 69.8973, Z -8.0000, A 0.000, B 0.000, C 0.000 }
gfCNCPoint5[25707] = {X 510.4795, Y 69.0822, Z -8.0000, A 0.000, B 0.000, C 0.000 }
gfCNCPoint5[25708] = {X 509.6267, Y 68.7047, Z -8.0000, A 0.000, B 0.000, C 0.000 }
gfCNCPoint5[25709] = {X 508.7892, Y 68.2944, Z -8.0000, A 0.000, B 0.000, C 0.000 }
gfCNCPoint5[25710] = {X 507.1695, Y 68.6594, Z -8.0000, A 0.000, B 0.000, C 0.000 }
gfCNCPoint5[25711] = {X 505.5286, Y 68.9119, Z -8.0000, A 0.000, B 0.000, C 0.000 }
gfCNCPoint5[25712] = {X 504.1110, Y 69.0379, Z -8.0000, A 0.000, B 0.000, C 0.000 }
gfCNCPoint5[25713] = {X 502.6885, Y 69.0800, Z -8.0000, A 0.000, B 0.000, C 0.000 }
gfCNCPoint5[25714] = {X 502.0391, Y 69.0800, Z -8.0000, A 0.000, B 0.000, C 0.000 }
gfCNCPoint5[25715] = {X 501.1779, Y 71.1312, Z -8.0000, A 0.000, B 0.000, C 0.000 }
gfCNCPoint5[25716] = {X 500.1614, Y 73.1101, Z -8.0000, A 0.000, B 0.000, C 0.000 }
gfCNCPoint5[25717] = {X 500.1614, Y 73.6952, Z -8.0000, A 0.000, B 0.000, C 0.000 }
gfCNCPoint5[25718] = {X 507.6811, Y 73.6952, Z -8.0000, A 0.000, B 0.000, C 0.000 }
gfCNCPoint5[25719] = {X 507.6811, Y 76.0952, Z -8.0000, A 0.000, B 0.000, C 0.000 }
gfCNCPoint5[25720] = {X 576.0967, Y 76.0952, Z -8.0000, A 0.000, B 0.000, C 0.000 }
gfCNCPoint5[25721] = {X 576.0967, Y 72.8902, Z -8.0000, A 0.000, B 0.000, C 0.000 }
gfCNCPoint5[25722] = {X 575.7179, Y 72.8147, Z -8.0000, A 0.000, B 0.000, C 0.000 }
gfCNCPoint5[25723] = {X 575.3401, Y 72.7341, Z -8.0000, A 0.000, B 0.000, C 0.000 }
gfCNCPoint5[25724] = {X 573.3201, Y 73.1034, Z -8.0000, A 0.000, B 0.000, C 0.000 }
gfCNCPoint5[25725] = {X 571.2786, Y 73.3258, Z -8.0000, A 0.000, B 0.000, C 0.000 }
gfCNCPoint5[25726] = {X 569.2264, Y 73.4000, Z -8.0000, A 0.000, B 0.000, C 0.000 }
gfCNCPoint5[25727] = {X 562.4443, Y 73.4000, Z -8.0000, A 0.000, B 0.000, C 0.000 }
gfCNCPoint5[25728] = {X 560.3342, Y 73.3215, Z -8.0000, A 0.000, B 0.000, C 0.000 }
gfCNCPoint5[25729] = {X 558.2358, Y 73.0864, Z -8.0000, A 0.000, B 0.000, C 0.000 }
gfCNCPoint5[25730] = {X 556.1606, Y 72.6961, Z -8.0000, A 0.000, B 0.000, C 0.000 }
gfCNCPoint5[25731] = {X 554.1202, Y 72.1527, Z -8.0000, A 0.000, B 0.000, C 0.000 }
gfCNCPoint5[25732] = {X 552.1258, Y 71.4592, Z -8.0000, A 0.000, B 0.000, C 0.000 }
gfCNCPoint5[25733] = {X 549.9769, Y 70.5171, Z -8.0000, A 0.000, B 0.000, C 0.000 }
gfCNCPoint5[25734] = {X 547.9131, Y 69.4009, Z -8.0000, A 0.000, B 0.000, C 0.000 }
gfCNCPoint5[25735] = {X 545.9485, Y 68.1182, Z -8.0000, A 0.000, B 0.000, C 0.000 }
gfCNCPoint5[25736] = {X 544.0965, Y 66.6776, Z -8.0000, A 0.000, B 0.000, C 0.000 }
gfCNCPoint5[25737] = {X 543.8508, Y 66.6788, Z -8.0000, A 0.000, B 0.000, C 0.000 }
gfCNCPoint5[25738] = {X 543.6051, Y 66.6773, Z -8.0000, A 0.000, B 0.000, C 0.000 }
gfCNCPoint5[25739] = {X 529.2669, Y 66.6775, Z -8.0000, A 0.000, B 0.000, C 0.000 }
gfCNCPoint5[25740] = {X 527.1796, Y 67.4799, Z -8.0000, A 0.000, B 0.000, C 0.000 }
gfCNCPoint5[25741] = {X 525.0211, Y 68.0647, Z -8.0000, A 0.000, B 0.000, C 0.000 }
gfCNCPoint5[25742] = {X 522.8141, Y 68.4256, Z -8.0000, A 0.000, B 0.000, C 0.000 }
gfCNCPoint5[25743] = {X 520.5818, Y 68.5589, Z -8.0000, A 0.000, B 0.000, C 0.000 }
gfCNCPoint5[25744] = {X 519.7998, Y 68.5591, Z -8.0000, A 0.000, B 0.000, C 0.000 }
gfCNCPoint5[25745] = {X 517.5593, Y 68.4430, Z -8.0000, A 0.000, B 0.000, C 0.000 }
gfCNCPoint5[25746] = {X 515.3429, Y 68.0961, Z -8.0000, A 0.000, B 0.000, C 0.000 }
gfCNCPoint5[25747] = {X 513.1742, Y 67.5219, Z -8.0000, A 0.000, B 0.000, C 0.000 }
gfCNCPoint5[25748] = {X 511.0764, Y 66.7267, Z -8.0000, A 0.000, B 0.000, C 0.000 }
gfCNCPoint5[25749] = {X 509.0720, Y 65.7189, Z -8.0000, A 0.000, B 0.000, C 0.000 }
gfCNCPoint5[25750] = {X 506.9797, Y 66.2511, Z -8.0000, A 0.000, B 0.000, C 0.000 }
gfCNCPoint5[25751] = {X 504.8448, Y 66.5725, Z -8.0000, A 0.000, B 0.000, C 0.000 }
gfCNCPoint5[25752] = {X 502.6885, Y 66.6800, Z -8.0000, A 0.000, B 0.000, C 0.000 }
gfCNCPoint5[25753] = {X 500.3217, Y 66.6800, Z -8.0000, A 0.000, B 0.000, C 0.000 }
gfCNCPoint5[25754] = {X 499.6233, Y 68.6748, Z -8.0000, A 0.000, B 0.000, C 0.000 }
gfCNCPoint5[25755] = {X 498.7681, Y 70.6075, Z -8.0000, A 0.000, B 0.000, C 0.000 }
gfCNCPoint5[25756] = {X 497.7614, Y 72.4659, Z -8.0000, A 0.000, B 0.000, C 0.000 }
gfCNCPoint5[25757] = {X 497.7614, Y 76.0952, Z -8.0000, A 0.000, B 0.000, C 0.000 }
gfCNCPoint5[25758] = {X 507.6811, Y 76.0952, Z -8.0000, A 0.000, B 0.000, C 0.000 }
gfCNCPoint5[25759] = {X 507.6811, Y 78.4952, Z -8.0000, A 0.000, B 0.000, C 0.000 }
gfCNCPoint5[25760] = {X 578.4967, Y 78.4952, Z -8.0000, A 0.000, B 0.000, C 0.000 }
gfCNCPoint5[25761] = {X 578.4967, Y 70.8313, Z -8.0000, A 0.000, B 0.000, C 0.000 }
gfCNCPoint5[25762] = {X 576.9098, Y 70.5998, Z -8.0000, A 0.000, B 0.000, C 0.000 }
gfCNCPoint5[25763] = {X 575.3401, Y 70.2710, Z -8.0000, A 0.000, B 0.000, C 0.000 }
gfCNCPoint5[25764] = {X 573.3236, Y 70.6751, Z -8.0000, A 0.000, B 0.000, C 0.000 }
gfCNCPoint5[25765] = {X 571.2815, Y 70.9187, Z -8.0000, A 0.000, B 0.000, C 0.000 }
gfCNCPoint5[25766] = {X 569.2264, Y 71.0000, Z -8.0000, A 0.000, B 0.000, C 0.000 }
gfCNCPoint5[25767] = {X 562.4443, Y 71.0000, Z -8.0000, A 0.000, B 0.000, C 0.000 }
gfCNCPoint5[25768] = {X 560.0515, Y 70.8897, Z -8.0000, A 0.000, B 0.000, C 0.000 }
gfCNCPoint5[25769] = {X 557.6790, Y 70.5596, Z -8.0000, A 0.000, B 0.000, C 0.000 }
gfCNCPoint5[25770] = {X 555.3469, Y 70.0125, Z -8.0000, A 0.000, B 0.000, C 0.000 }
gfCNCPoint5[25771] = {X 553.0751, Y 69.2532, Z -8.0000, A 0.000, B 0.000, C 0.000 }
gfCNCPoint5[25772] = {X 550.8828, Y 68.2880, Z -8.0000, A 0.000, B 0.000, C 0.000 }
gfCNCPoint5[25773] = {X 548.7887, Y 67.1252, Z -8.0000, A 0.000, B 0.000, C 0.000 }
gfCNCPoint5[25774] = {X 546.8104, Y 65.7745, Z -8.0000, A 0.000, B 0.000, C 0.000 }
gfCNCPoint5[25775] = {X 544.9648, Y 64.2476, Z -8.0000, A 0.000, B 0.000, C 0.000 }
gfCNCPoint5[25776] = {X 544.2927, Y 64.2741, Z -8.0000, A 0.000, B 0.000, C 0.000 }
gfCNCPoint5[25777] = {X 543.6200, Y 64.2773, Z -8.0000, A 0.000, B 0.000, C 0.000 }
gfCNCPoint5[25778] = {X 528.7420, Y 64.2775, Z -8.0000, A 0.000, B 0.000, C 0.000 }
gfCNCPoint5[25779] = {X 526.7883, Y 65.0792, Z -8.0000, A 0.000, B 0.000, C 0.000 }
gfCNCPoint5[25780] = {X 524.7590, Y 65.6641, Z -8.0000, A 0.000, B 0.000, C 0.000 }
gfCNCPoint5[25781] = {X 522.6783, Y 66.0254, Z -8.0000, A 0.000, B 0.000, C 0.000 }
gfCNCPoint5[25782] = {X 520.5707, Y 66.1589, Z -8.0000, A 0.000, B 0.000, C 0.000 }
gfCNCPoint5[25783] = {X 519.7998, Y 66.1591, Z -8.0000, A 0.000, B 0.000, C 0.000 }
gfCNCPoint5[25784] = {X 517.9641, Y 66.0715, Z -8.0000, A 0.000, B 0.000, C 0.000 }
gfCNCPoint5[25785] = {X 516.1450, Y 65.8096, Z -8.0000, A 0.000, B 0.000, C 0.000 }
gfCNCPoint5[25786] = {X 514.3592, Y 65.3756, Z -8.0000, A 0.000, B 0.000, C 0.000 }
gfCNCPoint5[25787] = {X 512.6228, Y 64.7735, Z -8.0000, A 0.000, B 0.000, C 0.000 }
gfCNCPoint5[25788] = {X 510.9516, Y 64.0089, Z -8.0000, A 0.000, B 0.000, C 0.000 }
gfCNCPoint5[25789] = {X 509.3609, Y 63.0886, Z -8.0000, A 0.000, B 0.000, C 0.000 }
gfCNCPoint5[25790] = {X 507.7389, Y 63.6068, Z -8.0000, A 0.000, B 0.000, C 0.000 }
gfCNCPoint5[25791] = {X 506.0774, Y 63.9798, Z -8.0000, A 0.000, B 0.000, C 0.000 }
gfCNCPoint5[25792] = {X 504.3896, Y 64.2048, Z -8.0000, A 0.000, B 0.000, C 0.000 }
gfCNCPoint5[25793] = {X 502.6885, Y 64.2800, Z -8.0000, A 0.000, B 0.000, C 0.000 }
gfCNCPoint5[25794] = {X 498.4791, Y 64.2800, Z -8.0000, A 0.000, B 0.000, C 0.000 }
gfCNCPoint5[25795] = {X 497.9418, Y 66.2499, Z -8.0000, A 0.000, B 0.000, C 0.000 }
gfCNCPoint5[25796] = {X 497.2395, Y 68.1673, Z -8.0000, A 0.000, B 0.000, C 0.000 }
gfCNCPoint5[25797] = {X 496.3773, Y 70.0182, Z -8.0000, A 0.000, B 0.000, C 0.000 }
gfCNCPoint5[25798] = {X 495.3614, Y 71.7895, Z -8.0000, A 0.000, B 0.000, C 0.000 }
gfCNCPoint5[25799] = {X 495.3615, Y 78.4952, Z -8.0000, A 0.000, B 0.000, C 0.000 }
gfCNCPoint5[25800] = {X 507.6811, Y 78.4952, Z -8.0000, A 0.000, B 0.000, C 0.000 }
gfCNCPoint5[25801] = {X 507.6811, Y 80.8952, Z -8.0000, A 0.000, B 0.000, C 0.000 }
gfCNCPoint5[25802] = {X 580.8967, Y 80.8952, Z -8.0000, A 0.000, B 0.000, C 0.000 }
gfCNCPoint5[25803] = {X 580.8967, Y 68.5934, Z -8.0000, A 0.000, B 0.000, C 0.000 }
gfCNCPoint5[25804] = {X 579.0253, Y 68.4747, Z -8.0000, A 0.000, B 0.000, C 0.000 }
gfCNCPoint5[25805] = {X 577.1692, Y 68.2078, Z -8.0000, A 0.000, B 0.000, C 0.000 }
gfCNCPoint5[25806] = {X 575.3401, Y 67.7943, Z -8.0000, A 0.000, B 0.000, C 0.000 }
gfCNCPoint5[25807] = {X 573.3283, Y 68.2408, Z -8.0000, A 0.000, B 0.000, C 0.000 }
gfCNCPoint5[25808] = {X 571.2852, Y 68.5100, Z -8.0000, A 0.000, B 0.000, C 0.000 }
gfCNCPoint5[25809] = {X 569.2264, Y 68.6000, Z -8.0000, A 0.000, B 0.000, C 0.000 }
gfCNCPoint5[25810] = {X 562.4443, Y 68.6000, Z -8.0000, A 0.000, B 0.000, C 0.000 }
gfCNCPoint5[25811] = {X 560.1445, Y 68.4877, Z -8.0000, A 0.000, B 0.000, C 0.000 }
gfCNCPoint5[25812] = {X 557.8667, Y 68.1518, Z -8.0000, A 0.000, B 0.000, C 0.000 }
gfCNCPoint5[25813] = {X 555.6324, Y 67.5955, Z -8.0000, A 0.000, B 0.000, C 0.000 }
gfCNCPoint5[25814] = {X 553.4629, Y 66.8242, Z -8.0000, A 0.000, B 0.000, C 0.000 }
gfCNCPoint5[25815] = {X 551.3790, Y 65.8451, Z -8.0000, A 0.000, B 0.000, C 0.000 }
gfCNCPoint5[25816] = {X 549.4003, Y 64.6676, Z -8.0000, A 0.000, B 0.000, C 0.000 }
gfCNCPoint5[25817] = {X 547.5458, Y 63.3029, Z -8.0000, A 0.000, B 0.000, C 0.000 }
gfCNCPoint5[25818] = {X 545.8332, Y 61.7640, Z -8.0000, A 0.000, B 0.000, C 0.000 }
gfCNCPoint5[25819] = {X 544.7364, Y 61.8564, Z -8.0000, A 0.000, B 0.000, C 0.000 }
gfCNCPoint5[25820] = {X 543.6358, Y 61.8773, Z -8.0000, A 0.000, B 0.000, C 0.000 }
gfCNCPoint5[25821] = {X 528.1818, Y 61.8775, Z -8.0000, A 0.000, B 0.000, C 0.000 }
gfCNCPoint5[25822] = {X 526.3714, Y 62.6781, Z -8.0000, A 0.000, B 0.000, C 0.000 }
gfCNCPoint5[25823] = {X 524.4803, Y 63.2633, Z -8.0000, A 0.000, B 0.000, C 0.000 }
gfCNCPoint5[25824] = {X 522.5341, Y 63.6252, Z -8.0000, A 0.000, B 0.000, C 0.000 }
gfCNCPoint5[25825] = {X 520.5590, Y 63.7589, Z -8.0000, A 0.000, B 0.000, C 0.000 }
gfCNCPoint5[25826] = {X 519.7998, Y 63.7591, Z -8.0000, A 0.000, B 0.000, C 0.000 }
gfCNCPoint5[25827] = {X 517.9902, Y 63.6618, Z -8.0000, A 0.000, B 0.000, C 0.000 }
gfCNCPoint5[25828] = {X 516.2015, Y 63.3711, Z -8.0000, A 0.000, B 0.000, C 0.000 }
gfCNCPoint5[25829] = {X 514.4543, Y 62.8904, Z -8.0000, A 0.000, B 0.000, C 0.000 }
gfCNCPoint5[25830] = {X 512.7687, Y 62.2251, Z -8.0000, A 0.000, B 0.000, C 0.000 }
gfCNCPoint5[25831] = {X 511.1641, Y 61.3829, Z -8.0000, A 0.000, B 0.000, C 0.000 }
gfCNCPoint5[25832] = {X 509.6590, Y 60.3735, Z -8.0000, A 0.000, B 0.000, C 0.000 }
gfCNCPoint5[25833] = {X 507.9866, Y 61.0270, Z -8.0000, A 0.000, B 0.000, C 0.000 }
gfCNCPoint5[25834] = {X 506.2542, Y 61.4991, Z -8.0000, A 0.000, B 0.000, C 0.000 }
gfCNCPoint5[25835] = {X 504.4815, Y 61.7845, Z -8.0000, A 0.000, B 0.000, C 0.000 }
gfCNCPoint5[25836] = {X 502.6885, Y 61.8800, Z -8.0000, A 0.000, B 0.000, C 0.000 }
gfCNCPoint5[25837] = {X 496.4789, Y 61.8800, Z -8.0000, A 0.000, B 0.000, C 0.000 }
gfCNCPoint5[25838] = {X 496.1193, Y 63.8328, Z -8.0000, A 0.000, B 0.000, C 0.000 }
gfCNCPoint5[25839] = {X 495.5825, Y 65.7446, Z -8.0000, A 0.000, B 0.000, C 0.000 }
gfCNCPoint5[25840] = {X 494.8730, Y 67.5992, Z -8.0000, A 0.000, B 0.000, C 0.000 }
gfCNCPoint5[25841] = {X 493.9969, Y 69.3811, Z -8.0000, A 0.000, B 0.000, C 0.000 }
gfCNCPoint5[25842] = {X 492.9614, Y 71.0754, Z -8.0000, A 0.000, B 0.000, C 0.000 }
gfCNCPoint5[25843] = {X 492.9615, Y 80.8952, Z -8.0000, A 0.000, B 0.000, C 0.000 }
gfCNCPoint5[25844] = {X 507.6811, Y 80.8952, Z -8.0000, A 0.000, B 0.000, C 0.000 }
gfCNCPoint5[25845] = {X 507.6811, Y 83.2952, Z -8.0000, A 0.000, B 0.000, C 0.000 }
gfCNCPoint5[25846] = {X 583.2967, Y 83.2952, Z -8.0000, A 0.000, B 0.000, C 0.000 }
gfCNCPoint5[25847] = {X 583.2967, Y 66.1198, Z -8.0000, A 0.000, B 0.000, C 0.000 }
gfCNCPoint5[25848] = {X 581.2873, Y 66.1993, Z -8.0000, A 0.000, B 0.000, C 0.000 }
gfCNCPoint5[25849] = {X 579.2794, Y 66.0882, Z -8.0000, A 0.000, B 0.000, C 0.000 }
gfCNCPoint5[25850] = {X 577.2910, Y 65.7873, Z -8.0000, A 0.000, B 0.000, C 0.000 }
gfCNCPoint5[25851] = {X 575.3401, Y 65.2993, Z -8.0000, A 0.000, B 0.000, C 0.000 }
gfCNCPoint5[25852] = {X 573.3348, Y 65.7981, Z -8.0000, A 0.000, B 0.000, C 0.000 }
gfCNCPoint5[25853] = {X 571.2904, Y 66.0993, Z -8.0000, A 0.000, B 0.000, C 0.000 }
gfCNCPoint5[25854] = {X 569.2264, Y 66.2000, Z -8.0000, A 0.000, B 0.000, C 0.000 }
gfCNCPoint5[25855] = {X 562.4443, Y 66.2000, Z -8.0000, A 0.000, B 0.000, C 0.000 }
gfCNCPoint5[25856] = {X 560.2305, Y 66.0841, Z -8.0000, A 0.000, B 0.000, C 0.000 }
gfCNCPoint5[25857] = {X 558.0409, Y 65.7377, Z -8.0000, A 0.000, B 0.000, C 0.000 }
gfCNCPoint5[25858] = {X 555.8995, Y 65.1645, Z -8.0000, A 0.000, B 0.000, C 0.000 }
gfCNCPoint5[25859] = {X 553.8296, Y 64.3708, Z -8.0000, A 0.000, B 0.000, C 0.000 }
gfCNCPoint5[25860] = {X 551.8539, Y 63.3653, Z -8.0000, A 0.000, B 0.000, C 0.000 }
gfCNCPoint5[25861] = {X 549.9940, Y 62.1590, Z -8.0000, A 0.000, B 0.000, C 0.000 }
gfCNCPoint5[25862] = {X 548.2703, Y 60.7651, Z -8.0000, A 0.000, B 0.000, C 0.000 }
gfCNCPoint5[25863] = {X 546.7015, Y 59.1988, Z -8.0000, A 0.000, B 0.000, C 0.000 }
gfCNCPoint5[25864] = {X 545.1846, Y 59.4188, Z -8.0000, A 0.000, B 0.000, C 0.000 }
gfCNCPoint5[25865] = {X 543.6529, Y 59.4773, Z -8.0000, A 0.000, B 0.000, C 0.000 }
gfCNCPoint5[25866] = {X 527.5780, Y 59.4775, Z -8.0000, A 0.000, B 0.000, C 0.000 }
gfCNCPoint5[25867] = {X 525.9207, Y 60.2778, Z -8.0000, A 0.000, B 0.000, C 0.000 }
gfCNCPoint5[25868] = {X 524.1760, Y 60.8637, Z -8.0000, A 0.000, B 0.000, C 0.000 }
gfCNCPoint5[25869] = {X 522.3716, Y 61.2260, Z -8.0000, A 0.000, B 0.000, C 0.000 }
gfCNCPoint5[25870] = {X 520.5360, Y 61.3590, Z -8.0000, A 0.000, B 0.000, C 0.000 }
gfCNCPoint5[25871] = {X 519.7998, Y 61.3591, Z -8.0000, A 0.000, B 0.000, C 0.000 }
gfCNCPoint5[25872] = {X 518.0043, Y 61.2474, Z -8.0000, A 0.000, B 0.000, C 0.000 }
gfCNCPoint5[25873] = {X 516.2365, Y 60.9138, Z -8.0000, A 0.000, B 0.000, C 0.000 }
gfCNCPoint5[25874] = {X 514.5237, Y 60.3637, Z -8.0000, A 0.000, B 0.000, C 0.000 }
gfCNCPoint5[25875] = {X 512.8923, Y 59.6054, Z -8.0000, A 0.000, B 0.000, C 0.000 }
gfCNCPoint5[25876] = {X 511.3676, Y 58.6507, Z -8.0000, A 0.000, B 0.000, C 0.000 }
gfCNCPoint5[25877] = {X 509.9730, Y 57.5142, Z -8.0000, A 0.000, B 0.000, C 0.000 }
gfCNCPoint5[25878] = {X 508.6156, Y 58.2113, Z -8.0000, A 0.000, B 0.000, C 0.000 }
gfCNCPoint5[25879] = {X 507.1924, Y 58.7617, Z -8.0000, A 0.000, B 0.000, C 0.000 }
gfCNCPoint5[25880] = {X 505.7192, Y 59.1593, Z -8.0000, A 0.000, B 0.000, C 0.000 }
gfCNCPoint5[25881] = {X 504.2123, Y 59.3996, Z -8.0000, A 0.000, B 0.000, C 0.000 }
gfCNCPoint5[25882] = {X 502.6885, Y 59.4800, Z -8.0000, A 0.000, B 0.000, C 0.000 }
gfCNCPoint5[25883] = {X 496.2450, Y 59.4800, Z -8.0000, A 0.000, B 0.000, C 0.000 }
gfCNCPoint5[25884] = {X 495.2580, Y 59.4463, Z -8.0000, A 0.000, B 0.000, C 0.000 }
gfCNCPoint5[25885] = {X 494.2756, Y 59.3454, Z -8.0000, A 0.000, B 0.000, C 0.000 }
gfCNCPoint5[25886] = {X 494.1342, Y 61.3003, Z -8.0000, A 0.000, B 0.000, C 0.000 }
gfCNCPoint5[25887] = {X 493.7952, Y 63.2306, Z -8.0000, A 0.000, B 0.000, C 0.000 }
gfCNCPoint5[25888] = {X 493.2618, Y 65.1166, Z -8.0000, A 0.000, B 0.000, C 0.000 }
gfCNCPoint5[25889] = {X 492.5398, Y 66.9386, Z -8.0000, A 0.000, B 0.000, C 0.000 }
gfCNCPoint5[25890] = {X 491.6365, Y 68.6780, Z -8.0000, A 0.000, B 0.000, C 0.000 }
gfCNCPoint5[25891] = {X 490.5613, Y 70.3166, Z -8.0000, A 0.000, B 0.000, C 0.000 }
gfCNCPoint5[25892] = {X 490.5616, Y 83.2952, Z -8.0000, A 0.000, B 0.000, C 0.000 }
gfCNCPoint5[25893] = {X 507.6811, Y 83.2952, Z -8.0000, A 0.000, B 0.000, C 0.000 }
gfCNCPoint5[25894] = {X 507.6811, Y 85.6952, Z -8.0000, A 0.000, B 0.000, C 0.000 }
gfCNCPoint5[25895] = {X 585.6967, Y 85.6952, Z -8.0000, A 0.000, B 0.000, C 0.000 }
gfCNCPoint5[25896] = {X 585.6967, Y 63.3150, Z -8.0000, A 0.000, B 0.000, C 0.000 }
gfCNCPoint5[25897] = {X 584.3997, Y 63.5678, Z -8.0000, A 0.000, B 0.000, C 0.000 }
gfCNCPoint5[25898] = {X 583.0881, Y 63.7288, Z -8.0000, A 0.000, B 0.000, C 0.000 }
gfCNCPoint5[25899] = {X 581.1243, Y 63.7971, Z -8.0000, A 0.000, B 0.000, C 0.000 }
gfCNCPoint5[25900] = {X 579.1642, Y 63.6600, Z -8.0000, A 0.000, B 0.000, C 0.000 }
gfCNCPoint5[25901] = {X 577.2291, Y 63.3192, Z -8.0000, A 0.000, B 0.000, C 0.000 }
gfCNCPoint5[25902] = {X 575.3401, Y 62.7781, Z -8.0000, A 0.000, B 0.000, C 0.000 }
gfCNCPoint5[25903] = {X 573.3441, Y 63.3435, Z -8.0000, A 0.000, B 0.000, C 0.000 }
gfCNCPoint5[25904] = {X 571.2979, Y 63.6855, Z -8.0000, A 0.000, B 0.000, C 0.000 }
gfCNCPoint5[25905] = {X 569.2264, Y 63.8000, Z -8.0000, A 0.000, B 0.000, C 0.000 }
gfCNCPoint5[25906] = {X 562.4443, Y 63.8000, Z -8.0000, A 0.000, B 0.000, C 0.000 }
gfCNCPoint5[25907] = {X 560.5409, Y 63.7034, Z -8.0000, A 0.000, B 0.000, C 0.000 }
gfCNCPoint5[25908] = {X 558.6571, Y 63.4146, Z -8.0000, A 0.000, B 0.000, C 0.000 }
gfCNCPoint5[25909] = {X 556.8122, Y 62.9365, Z -8.0000, A 0.000, B 0.000, C 0.000 }
gfCNCPoint5[25910] = {X 555.0252, Y 62.2742, Z -8.0000, A 0.000, B 0.000, C 0.000 }
gfCNCPoint5[25911] = {X 553.3144, Y 61.4343, Z -8.0000, A 0.000, B 0.000, C 0.000 }
gfCNCPoint5[25912] = {X 551.6975, Y 60.4255, Z -8.0000, A 0.000, B 0.000, C 0.000 }
gfCNCPoint5[25913] = {X 550.1910, Y 59.2582, Z -8.0000, A 0.000, B 0.000, C 0.000 }
gfCNCPoint5[25914] = {X 548.8104, Y 57.9444, Z -8.0000, A 0.000, B 0.000, C 0.000 }
gfCNCPoint5[25915] = {X 547.5699, Y 56.4975, Z -8.0000, A 0.000, B 0.000, C 0.000 }
gfCNCPoint5[25916] = {X 546.2942, Y 56.8326, Z -8.0000, A 0.000, B 0.000, C 0.000 }
gfCNCPoint5[25917] = {X 544.9895, Y 57.0266, Z -8.0000, A 0.000, B 0.000, C 0.000 }
gfCNCPoint5[25918] = {X 543.6714, Y 57.0773, Z -8.0000, A 0.000, B 0.000, C 0.000 }
gfCNCPoint5[25919] = {X 526.9186, Y 57.0775, Z -8.0000, A 0.000, B 0.000, C 0.000 }
gfCNCPoint5[25920] = {X 525.4330, Y 57.8758, Z -8.0000, A 0.000, B 0.000, C 0.000 }
gfCNCPoint5[25921] = {X 523.8517, Y 58.4622, Z -8.0000, A 0.000, B 0.000, C 0.000 }
gfCNCPoint5[25922] = {X 522.2047, Y 58.8255, Z -8.0000, A 0.000, B 0.000, C 0.000 }
gfCNCPoint5[25923] = {X 520.5235, Y 58.9590, Z -8.0000, A 0.000, B 0.000, C 0.000 }
gfCNCPoint5[25924] = {X 519.7998, Y 58.9591, Z -8.0000, A 0.000, B 0.000, C 0.000 }
gfCNCPoint5[25925] = {X 518.2467, Y 58.8589, Z -8.0000, A 0.000, B 0.000, C 0.000 }
gfCNCPoint5[25926] = {X 516.7195, Y 58.5598, Z -8.0000, A 0.000, B 0.000, C 0.000 }
gfCNCPoint5[25927] = {X 515.2433, Y 58.0668, Z -8.0000, A 0.000, B 0.000, C 0.000 }
gfCNCPoint5[25928] = {X 513.8428, Y 57.3882, Z -8.0000, A 0.000, B 0.000, C 0.000 }
gfCNCPoint5[25929] = {X 512.5411, Y 56.5351, Z -8.0000, A 0.000, B 0.000, C 0.000 }
gfCNCPoint5[25930] = {X 511.3600, Y 55.5218, Z -8.0000, A 0.000, B 0.000, C 0.000 }
gfCNCPoint5[25931] = {X 510.3189, Y 54.3650, Z -8.0000, A 0.000, B 0.000, C 0.000 }
gfCNCPoint5[25932] = {X 508.9711, Y 55.3177, Z -8.0000, A 0.000, B 0.000, C 0.000 }
gfCNCPoint5[25933] = {X 507.5060, Y 56.0778, Z -8.0000, A 0.000, B 0.000, C 0.000 }
gfCNCPoint5[25934] = {X 505.9510, Y 56.6311, Z -8.0000, A 0.000, B 0.000, C 0.000 }
gfCNCPoint5[25935] = {X 504.3351, Y 56.9672, Z -8.0000, A 0.000, B 0.000, C 0.000 }
gfCNCPoint5[25936] = {X 502.6885, Y 57.0800, Z -8.0000, A 0.000, B 0.000, C 0.000 }
gfCNCPoint5[25937] = {X 496.2450, Y 57.0800, Z -8.0000, A 0.000, B 0.000, C 0.000 }
gfCNCPoint5[25938] = {X 495.4216, Y 57.0519, Z -8.0000, A 0.000, B 0.000, C 0.000 }
gfCNCPoint5[25939] = {X 494.6020, Y 56.9677, Z -8.0000, A 0.000, B 0.000, C 0.000 }
gfCNCPoint5[25940] = {X 493.1719, Y 56.6826, Z -8.0000, A 0.000, B 0.000, C 0.000 }
gfCNCPoint5[25941] = {X 491.7866, Y 56.2272, Z -8.0000, A 0.000, B 0.000, C 0.000 }
gfCNCPoint5[25942] = {X 491.8566, Y 57.1124, Z -8.0000, A 0.000, B 0.000, C 0.000 }
gfCNCPoint5[25943] = {X 491.8800, Y 58.0000, Z -8.0000, A 0.000, B 0.000, C 0.000 }
gfCNCPoint5[25944] = {X 491.8794, Y 59.0735, Z -8.0000, A 0.000, B 0.000, C 0.000 }
gfCNCPoint5[25945] = {X 491.8782, Y 59.1839, Z -8.0000, A 0.000, B 0.000, C 0.000 }
gfCNCPoint5[25946] = {X 491.8762, Y 59.2942, Z -8.0000, A 0.000, B 0.000, C 0.000 }
gfCNCPoint5[25947] = {X 491.7364, Y 61.1315, Z -8.0000, A 0.000, B 0.000, C 0.000 }
gfCNCPoint5[25948] = {X 491.3971, Y 62.9426, Z -8.0000, A 0.000, B 0.000, C 0.000 }
gfCNCPoint5[25949] = {X 490.8625, Y 64.7059, Z -8.0000, A 0.000, B 0.000, C 0.000 }
gfCNCPoint5[25950] = {X 490.1389, Y 66.4005, Z -8.0000, A 0.000, B 0.000, C 0.000 }
gfCNCPoint5[25951] = {X 489.2349, Y 68.0060, Z -8.0000, A 0.000, B 0.000, C 0.000 }
gfCNCPoint5[25952] = {X 488.1613, Y 69.5035, Z -8.0000, A 0.000, B 0.000, C 0.000 }
gfCNCPoint5[25953] = {X 488.1616, Y 85.6952, Z -8.0000, A 0.000, B 0.000, C 0.000 }
gfCNCPoint5[25954] = {X 507.6811, Y 85.6952, Z -8.0000, A 0.000, B 0.000, C 0.000 }
gfCNCPoint5[25955] = {X 507.6811, Y 88.0952, Z -8.0000, A 0.000, B 0.000, C 0.000 }
gfCNCPoint5[25956] = {X 588.0967, Y 88.0952, Z -8.0000, A 0.000, B 0.000, C 0.000 }
gfCNCPoint5[25957] = {X 588.0967, Y 60.4645, Z -8.0000, A 0.000, B 0.000, C 0.000 }
gfCNCPoint5[25958] = {X 587.7999, Y 60.3565, Z -8.0000, A 0.000, B 0.000, C 0.000 }
gfCNCPoint5[25959] = {X 587.5052, Y 60.2427, Z -8.0000, A 0.000, B 0.000, C 0.000 }
gfCNCPoint5[25960] = {X 586.3439, Y 60.6540, Z -8.0000, A 0.000, B 0.000, C 0.000 }
gfCNCPoint5[25961] = {X 585.1551, Y 60.9769, Z -8.0000, A 0.000, B 0.000, C 0.000 }
gfCNCPoint5[25962] = {X 583.5154, Y 61.2699, Z -8.0000, A 0.000, B 0.000, C 0.000 }
gfCNCPoint5[25963] = {X 581.8544, Y 61.3951, Z -8.0000, A 0.000, B 0.000, C 0.000 }
gfCNCPoint5[25964] = {X 580.1893, Y 61.3512, Z -8.0000, A 0.000, B 0.000, C 0.000 }
gfCNCPoint5[25965] = {X 578.5373, Y 61.1386, Z -8.0000, A 0.000, B 0.000, C 0.000 }
gfCNCPoint5[25966] = {X 576.9153, Y 60.7595, Z -8.0000, A 0.000, B 0.000, C 0.000 }
gfCNCPoint5[25967] = {X 575.3401, Y 60.2178, Z -8.0000, A 0.000, B 0.000, C 0.000 }
gfCNCPoint5[25968] = {X 573.8611, Y 60.7315, Z -8.0000, A 0.000, B 0.000, C 0.000 }
gfCNCPoint5[25969] = {X 572.3399, Y 61.1017, Z -8.0000, A 0.000, B 0.000, C 0.000 }
gfCNCPoint5[25970] = {X 570.7903, Y 61.3253, Z -8.0000, A 0.000, B 0.000, C 0.000 }
gfCNCPoint5[25971] = {X 569.2264, Y 61.4000, Z -8.0000, A 0.000, B 0.000, C 0.000 }
gfCNCPoint5[25972] = {X 562.4443, Y 61.4000, Z -8.0000, A 0.000, B 0.000, C 0.000 }
gfCNCPoint5[25973] = {X 560.5830, Y 61.2940, Z -8.0000, A 0.000, B 0.000, C 0.000 }
gfCNCPoint5[25974] = {X 558.7457, Y 60.9775, Z -8.0000, A 0.000, B 0.000, C 0.000 }
gfCNCPoint5[25975] = {X 556.9562, Y 60.4545, Z -8.0000, A 0.000, B 0.000, C 0.000 }
gfCNCPoint5[25976] = {X 555.2377, Y 59.7318, Z -8.0000, A 0.000, B 0.000, C 0.000 }
gfCNCPoint5[25977] = {X 553.6123, Y 58.8187, Z -8.0000, A 0.000, B 0.000, C 0.000 }
gfCNCPoint5[25978] = {X 552.1010, Y 57.7270, Z -8.0000, A 0.000, B 0.000, C 0.000 }
gfCNCPoint5[25979] = {X 550.7234, Y 56.4708, Z -8.0000, A 0.000, B 0.000, C 0.000 }
gfCNCPoint5[25980] = {X 549.4972, Y 55.0665, Z -8.0000, A 0.000, B 0.000, C 0.000 }
gfCNCPoint5[25981] = {X 548.4384, Y 53.5320, Z -8.0000, A 0.000, B 0.000, C 0.000 }
gfCNCPoint5[25982] = {X 547.3164, Y 54.0437, Z -8.0000, A 0.000, B 0.000, C 0.000 }
gfCNCPoint5[25983] = {X 546.1385, Y 54.4087, Z -8.0000, A 0.000, B 0.000, C 0.000 }
gfCNCPoint5[25984] = {X 544.9238, Y 54.6210, Z -8.0000, A 0.000, B 0.000, C 0.000 }
gfCNCPoint5[25985] = {X 543.6919, Y 54.6773, Z -8.0000, A 0.000, B 0.000, C 0.000 }
gfCNCPoint5[25986] = {X 526.1845, Y 54.6775, Z -8.0000, A 0.000, B 0.000, C 0.000 }
gfCNCPoint5[25987] = {X 524.8900, Y 55.4740, Z -8.0000, A 0.000, B 0.000, C 0.000 }
gfCNCPoint5[25988] = {X 523.4883, Y 56.0616, Z -8.0000, A 0.000, B 0.000, C 0.000 }
gfCNCPoint5[25989] = {X 522.0128, Y 56.4262, Z -8.0000, A 0.000, B 0.000, C 0.000 }
gfCNCPoint5[25990] = {X 520.4987, Y 56.5591, Z -8.0000, A 0.000, B 0.000, C 0.000 }
gfCNCPoint5[25991] = {X 519.7998, Y 56.5591, Z -8.0000, A 0.000, B 0.000, C 0.000 }
gfCNCPoint5[25992] = {X 518.3493, Y 56.4498, Z -8.0000, A 0.000, B 0.000, C 0.000 }
gfCNCPoint5[25993] = {X 516.9316, Y 56.1244, Z -8.0000, A 0.000, B 0.000, C 0.000 }
gfCNCPoint5[25994] = {X 515.5787, Y 55.5903, Z -8.0000, A 0.000, B 0.000, C 0.000 }
gfCNCPoint5[25995] = {X 514.3210, Y 54.8595, Z -8.0000, A 0.000, B 0.000, C 0.000 }
gfCNCPoint5[25996] = {X 513.1871, Y 53.9484, Z -8.0000, A 0.000, B 0.000, C 0.000 }
gfCNCPoint5[25997] = {X 512.2025, Y 52.8778, Z -8.0000, A 0.000, B 0.000, C 0.000 }
gfCNCPoint5[25998] = {X 511.3855, Y 51.6648, Z -8.0000, A 0.000, B 0.000, C 0.000 }
gfCNCPoint5[25999] = {X 510.7606, Y 50.3426, Z -8.0000, A 0.000, B 0.000, C 0.000 }
gfCNCPoint5[26000] = {X 509.8636, Y 51.4977, Z -8.0000, A 0.000, B 0.000, C 0.000 }
gfCNCPoint5[26001] = {X 508.8029, Y 52.5044, Z -8.0000, A 0.000, B 0.000, C 0.000 }
gfCNCPoint5[26002] = {X 507.7229, Y 53.2678, Z -8.0000, A 0.000, B 0.000, C 0.000 }
gfCNCPoint5[26003] = {X 506.5489, Y 53.8769, Z -8.0000, A 0.000, B 0.000, C 0.000 }
gfCNCPoint5[26004] = {X 505.3028, Y 54.3203, Z -8.0000, A 0.000, B 0.000, C 0.000 }
gfCNCPoint5[26005] = {X 504.0080, Y 54.5896, Z -8.0000, A 0.000, B 0.000, C 0.000 }
gfCNCPoint5[26006] = {X 502.6885, Y 54.6800, Z -8.0000, A 0.000, B 0.000, C 0.000 }
gfCNCPoint5[26007] = {X 496.2450, Y 54.6800, Z -8.0000, A 0.000, B 0.000, C 0.000 }
gfCNCPoint5[26008] = {X 495.0285, Y 54.6033, Z -8.0000, A 0.000, B 0.000, C 0.000 }
gfCNCPoint5[26009] = {X 493.8313, Y 54.3742, Z -8.0000, A 0.000, B 0.000, C 0.000 }
gfCNCPoint5[26010] = {X 492.6724, Y 53.9966, Z -8.0000, A 0.000, B 0.000, C 0.000 }
gfCNCPoint5[26011] = {X 491.4451, Y 53.4062, Z -8.0000, A 0.000, B 0.000, C 0.000 }
gfCNCPoint5[26012] = {X 490.3129, Y 52.6493, Z -8.0000, A 0.000, B 0.000, C 0.000 }
gfCNCPoint5[26013] = {X 489.2980, Y 51.7410, Z -8.0000, A 0.000, B 0.000, C 0.000 }
gfCNCPoint5[26014] = {X 488.8683, Y 52.1573, Z -8.0000, A 0.000, B 0.000, C 0.000 }
gfCNCPoint5[26015] = {X 488.4137, Y 52.5463, Z -8.0000, A 0.000, B 0.000, C 0.000 }
gfCNCPoint5[26016] = {X 488.8649, Y 53.8245, Z -8.0000, A 0.000, B 0.000, C 0.000 }
gfCNCPoint5[26017] = {X 489.1946, Y 55.1393, Z -8.0000, A 0.000, B 0.000, C 0.000 }
gfCNCPoint5[26018] = {X 489.3999, Y 56.4792, Z -8.0000, A 0.000, B 0.000, C 0.000 }
gfCNCPoint5[26019] = {X 489.4600, Y 57.2386, Z -8.0000, A 0.000, B 0.000, C 0.000 }
gfCNCPoint5[26020] = {X 489.4800, Y 58.0000, Z -8.0000, A 0.000, B 0.000, C 0.000 }
gfCNCPoint5[26021] = {X 489.4795, Y 59.0537, Z -8.0000, A 0.000, B 0.000, C 0.000 }
gfCNCPoint5[26022] = {X 489.3596, Y 60.7975, Z -8.0000, A 0.000, B 0.000, C 0.000 }
gfCNCPoint5[26023] = {X 489.0304, Y 62.5141, Z -8.0000, A 0.000, B 0.000, C 0.000 }
gfCNCPoint5[26024] = {X 488.4969, Y 64.1786, Z -8.0000, A 0.000, B 0.000, C 0.000 }
gfCNCPoint5[26025] = {X 487.7666, Y 65.7667, Z -8.0000, A 0.000, B 0.000, C 0.000 }
gfCNCPoint5[26026] = {X 486.8503, Y 67.2552, Z -8.0000, A 0.000, B 0.000, C 0.000 }
gfCNCPoint5[26027] = {X 485.7613, Y 68.6224, Z -8.0000, A 0.000, B 0.000, C 0.000 }
gfCNCPoint5[26028] = {X 485.7616, Y 87.3810, Z -8.0000, A 0.000, B 0.000, C 0.000 }
gfCNCPoint5[26029] = {X 486.0689, Y 87.7332, Z -8.0000, A 0.000, B 0.000, C 0.000 }
gfCNCPoint5[26030] = {X 486.3646, Y 88.0952, Z -8.0000, A 0.000, B 0.000, C 0.000 }
gfCNCPoint5[26031] = {X 507.6811, Y 88.0952, Z -8.0000, A 0.000, B 0.000, C 0.000 }
gfCNCPoint5[26032] = {X 507.6811, Y 90.4952, Z -8.0000, A 0.000, B 0.000, C 0.000 }
gfCNCPoint5[26033] = {X 590.4967, Y 90.4952, Z -8.0000, A 0.000, B 0.000, C 0.000 }
gfCNCPoint5[26034] = {X 590.4967, Y 58.6615, Z -8.0000, A 0.000, B 0.000, C 0.000 }
gfCNCPoint5[26035] = {X 588.9715, Y 58.2279, Z -8.0000, A 0.000, B 0.000, C 0.000 }
gfCNCPoint5[26036] = {X 587.5052, Y 57.6246, Z -8.0000, A 0.000, B 0.000, C 0.000 }
gfCNCPoint5[26037] = {X 585.8387, Y 58.2956, Z -8.0000, A 0.000, B 0.000, C 0.000 }
gfCNCPoint5[26038] = {X 584.0999, Y 58.7477, Z -8.0000, A 0.000, B 0.000, C 0.000 }
gfCNCPoint5[26039] = {X 582.3176, Y 58.9733, Z -8.0000, A 0.000, B 0.000, C 0.000 }
gfCNCPoint5[26040] = {X 580.5210, Y 58.9689, Z -8.0000, A 0.000, B 0.000, C 0.000 }
gfCNCPoint5[26041] = {X 578.7398, Y 58.7344, Z -8.0000, A 0.000, B 0.000, C 0.000 }
gfCNCPoint5[26042] = {X 577.0034, Y 58.2738, Z -8.0000, A 0.000, B 0.000, C 0.000 }
gfCNCPoint5[26043] = {X 575.3401, Y 57.5945, Z -8.0000, A 0.000, B 0.000, C 0.000 }
gfCNCPoint5[26044] = {X 573.8813, Y 58.2035, Z -8.0000, A 0.000, B 0.000, C 0.000 }
gfCNCPoint5[26045] = {X 572.3630, Y 58.6441, Z -8.0000, A 0.000, B 0.000, C 0.000 }
gfCNCPoint5[26046] = {X 570.8048, Y 58.9107, Z -8.0000, A 0.000, B 0.000, C 0.000 }
gfCNCPoint5[26047] = {X 569.2264, Y 59.0000, Z -8.0000, A 0.000, B 0.000, C 0.000 }
gfCNCPoint5[26048] = {X 562.4443, Y 59.0000, Z -8.0000, A 0.000, B 0.000, C 0.000 }
gfCNCPoint5[26049] = {X 560.6578, Y 58.8855, Z -8.0000, A 0.000, B 0.000, C 0.000 }
gfCNCPoint5[26050] = {X 558.9005, Y 58.5440, Z -8.0000, A 0.000, B 0.000, C 0.000 }
gfCNCPoint5[26051] = {X 557.2011, Y 57.9811, Z -8.0000, A 0.000, B 0.000, C 0.000 }
gfCNCPoint5[26052] = {X 555.5875, Y 57.2059, Z -8.0000, A 0.000, B 0.000, C 0.000 }
gfCNCPoint5[26053] = {X 554.0859, Y 56.2311, Z -8.0000, A 0.000, B 0.000, C 0.000 }
gfCNCPoint5[26054] = {X 552.7211, Y 55.0727, Z -8.0000, A 0.000, B 0.000, C 0.000 }
gfCNCPoint5[26055] = {X 551.5152, Y 53.7496, Z -8.0000, A 0.000, B 0.000, C 0.000 }
gfCNCPoint5[26056] = {X 550.4880, Y 52.2834, Z -8.0000, A 0.000, B 0.000, C 0.000 }
gfCNCPoint5[26057] = {X 549.8382, Y 51.0898, Z -8.0000, A 0.000, B 0.000, C 0.000 }
gfCNCPoint5[26058] = {X 549.3071, Y 49.8388, Z -8.0000, A 0.000, B 0.000, C 0.000 }
gfCNCPoint5[26059] = {X 548.3758, Y 50.7157, Z -8.0000, A 0.000, B 0.000, C 0.000 }
gfCNCPoint5[26060] = {X 547.3055, Y 51.4162, Z -8.0000, A 0.000, B 0.000, C 0.000 }
gfCNCPoint5[26061] = {X 546.1638, Y 51.9072, Z -8.0000, A 0.000, B 0.000, C 0.000 }
gfCNCPoint5[26062] = {X 544.9553, Y 52.1971, Z -8.0000, A 0.000, B 0.000, C 0.000 }
gfCNCPoint5[26063] = {X 543.7151, Y 52.2773, Z -8.0000, A 0.000, B 0.000, C 0.000 }
gfCNCPoint5[26064] = {X 525.3426, Y 52.2775, Z -8.0000, A 0.000, B 0.000, C 0.000 }
gfCNCPoint5[26065] = {X 524.2751, Y 53.0689, Z -8.0000, A 0.000, B 0.000, C 0.000 }
gfCNCPoint5[26066] = {X 523.0839, Y 53.6577, Z -8.0000, A 0.000, B 0.000, C 0.000 }
gfCNCPoint5[26067] = {X 521.8068, Y 54.0250, Z -8.0000, A 0.000, B 0.000, C 0.000 }
gfCNCPoint5[26068] = {X 520.4848, Y 54.1591, Z -8.0000, A 0.000, B 0.000, C 0.000 }
gfCNCPoint5[26069] = {X 519.7998, Y 54.1591, Z -8.0000, A 0.000, B 0.000, C 0.000 }
gfCNCPoint5[26070] = {X 518.5529, Y 54.0515, Z -8.0000, A 0.000, B 0.000, C 0.000 }
gfCNCPoint5[26071] = {X 517.3428, Y 53.7320, Z -8.0000, A 0.000, B 0.000, C 0.000 }
gfCNCPoint5[26072] = {X 516.2054, Y 53.2099, Z -8.0000, A 0.000, B 0.000, C 0.000 }
gfCNCPoint5[26073] = {X 515.1742, Y 52.5007, Z -8.0000, A 0.000, B 0.000, C 0.000 }
gfCNCPoint5[26074] = {X 514.2797, Y 51.6254, Z -8.0000, A 0.000, B 0.000, C 0.000 }
gfCNCPoint5[26075] = {X 513.5483, Y 50.6098, Z -8.0000, A 0.000, B 0.000, C 0.000 }
gfCNCPoint5[26076] = {X 513.0017, Y 49.4839, Z -8.0000, A 0.000, B 0.000, C 0.000 }
gfCNCPoint5[26077] = {X 512.7353, Y 48.6374, Z -8.0000, A 0.000, B 0.000, C 0.000 }
gfCNCPoint5[26078] = {X 512.5739, Y 47.7649, Z -8.0000, A 0.000, B 0.000, C 0.000 }
gfCNCPoint5[26079] = {X 512.5198, Y 46.8791, Z -8.0000, A 0.000, B 0.000, C 0.000 }
gfCNCPoint5[26080] = {X 512.5198, Y 39.9011, Z -8.0000, A 0.000, B 0.000, C 0.000 }
gfCNCPoint5[26081] = {X 512.5808, Y 38.9602, Z -8.0000, A 0.000, B 0.000, C 0.000 }
gfCNCPoint5[26082] = {X 512.7630, Y 38.0352, Z -8.0000, A 0.000, B 0.000, C 0.000 }
gfCNCPoint5[26083] = {X 513.0631, Y 37.1414, Z -8.0000, A 0.000, B 0.000, C 0.000 }
gfCNCPoint5[26084] = {X 513.5588, Y 36.1529, Z -8.0000, A 0.000, B 0.000, C 0.000 }
gfCNCPoint5[26085] = {X 514.1985, Y 35.2509, Z -8.0000, A 0.000, B 0.000, C 0.000 }
gfCNCPoint5[26086] = {X 514.9674, Y 34.4562, Z -8.0000, A 0.000, B 0.000, C 0.000 }
gfCNCPoint5[26087] = {X 515.8478, Y 33.7872, Z -8.0000, A 0.000, B 0.000, C 0.000 }
gfCNCPoint5[26088] = {X 513.2421, Y 29.7560, Z -8.0000, A 0.000, B 0.000, C 0.000 }
gfCNCPoint5[26089] = {X 513.5223, Y 29.5803, Z -8.0000, A 0.000, B 0.000, C 0.000 }
gfCNCPoint5[26090] = {X 513.8071, Y 29.4123, Z -8.0000, A 0.000, B 0.000, C 0.000 }
gfCNCPoint5[26091] = {X 513.8074, Y 27.6761, Z -8.0000, A 0.000, B 0.000, C 0.000 }
gfCNCPoint5[26092] = {X 513.5223, Y 27.5016, Z -8.0000, A 0.000, B 0.000, C 0.000 }
gfCNCPoint5[26093] = {X 513.2421, Y 27.3193, Z -8.0000, A 0.000, B 0.000, C 0.000 }
gfCNCPoint5[26094] = {X 513.2421, Y 29.7560, Z -8.0000, A 0.000, B 0.000, C 0.000 }
gfCNCPoint5[26095] = {X 514.5450, Y 31.7716, Z -8.0000, A 0.000, B 0.000, C 0.000 }
gfCNCPoint5[26096] = {X 515.3551, Y 31.3018, Z -8.0000, A 0.000, B 0.000, C 0.000 }
gfCNCPoint5[26097] = {X 516.2069, Y 30.9126, Z -8.0000, A 0.000, B 0.000, C 0.000 }
gfCNCPoint5[26098] = {X 516.2077, Y 26.2050, Z -8.0000, A 0.000, B 0.000, C 0.000 }
gfCNCPoint5[26099] = {X 515.3721, Y 25.8045, Z -8.0000, A 0.000, B 0.000, C 0.000 }
gfCNCPoint5[26100] = {X 514.5786, Y 25.3259, Z -8.0000, A 0.000, B 0.000, C 0.000 }
gfCNCPoint5[26101] = {X 513.5955, Y 24.5712, Z -8.0000, A 0.000, B 0.000, C 0.000 }
gfCNCPoint5[26102] = {X 512.7168, Y 23.6972, Z -8.0000, A 0.000, B 0.000, C 0.000 }
gfCNCPoint5[26103] = {X 511.9571, Y 22.7180, Z -8.0000, A 0.000, B 0.000, C 0.000 }
gfCNCPoint5[26104] = {X 511.3287, Y 21.6498, Z -8.0000, A 0.000, B 0.000, C 0.000 }
gfCNCPoint5[26105] = {X 510.8419, Y 20.5101, Z -8.0000, A 0.000, B 0.000, C 0.000 }
gfCNCPoint5[26106] = {X 510.8423, Y 36.2316, Z -8.0000, A 0.000, B 0.000, C 0.000 }
gfCNCPoint5[26107] = {X 511.5014, Y 34.9173, Z -8.0000, A 0.000, B 0.000, C 0.000 }
gfCNCPoint5[26108] = {X 512.3519, Y 33.7179, Z -8.0000, A 0.000, B 0.000, C 0.000 }
gfCNCPoint5[26109] = {X 513.3743, Y 32.6612, Z -8.0000, A 0.000, B 0.000, C 0.000 }
gfCNCPoint5[26110] = {X 514.5450, Y 31.7716, Z -8.0000, A 0.000, B 0.000, C 0.000 }
gfCNCPoint5[26111] = {X 515.8478, Y 33.7872, Z -8.0000, A 0.000, B 0.000, C 0.000 }
gfCNCPoint5[26112] = {X 516.7441, Y 33.2934, Z -8.0000, A 0.000, B 0.000, C 0.000 }
gfCNCPoint5[26113] = {X 517.7008, Y 32.9302, Z -8.0000, A 0.000, B 0.000, C 0.000 }
gfCNCPoint5[26114] = {X 518.6990, Y 32.7048, Z -8.0000, A 0.000, B 0.000, C 0.000 }
gfCNCPoint5[26115] = {X 518.6299, Y 32.1290, Z -8.0000, A 0.000, B 0.000, C 0.000 }
gfCNCPoint5[26116] = {X 518.6068, Y 31.5495, Z -8.0000, A 0.000, B 0.000, C 0.000 }
gfCNCPoint5[26117] = {X 518.6080, Y 24.4373, Z -8.0000, A 0.000, B 0.000, C 0.000 }
gfCNCPoint5[26118] = {X 517.3914, Y 24.0941, Z -8.0000, A 0.000, B 0.000, C 0.000 }
gfCNCPoint5[26119] = {X 516.2525, Y 23.5456, Z -8.0000, A 0.000, B 0.000, C 0.000 }
gfCNCPoint5[26120] = {X 515.2257, Y 22.8083, Z -8.0000, A 0.000, B 0.000, C 0.000 }
gfCNCPoint5[26121] = {X 514.3419, Y 21.9045, Z -8.0000, A 0.000, B 0.000, C 0.000 }
gfCNCPoint5[26122] = {X 513.6278, Y 20.8615, Z -8.0000, A 0.000, B 0.000, C 0.000 }
gfCNCPoint5[26123] = {X 513.1048, Y 19.7107, Z -8.0000, A 0.000, B 0.000, C 0.000 }
gfCNCPoint5[26124] = {X 512.7938, Y 18.5159, Z -8.0000, A 0.000, B 0.000, C 0.000 }
gfCNCPoint5[26125] = {X 512.6891, Y 17.2857, Z -8.0000, A 0.000, B 0.000, C 0.000 }
gfCNCPoint5[26126] = {X 512.6891, Y 10.3077, Z -8.0000, A 0.000, B 0.000, C 0.000 }
gfCNCPoint5[26127] = {X 512.7002, Y 9.9056, Z -8.0000, A 0.000, B 0.000, C 0.000 }
gfCNCPoint5[26128] = {X 512.7335, Y 9.5048, Z -8.0000, A 0.000, B 0.000, C 0.000 }
gfCNCPoint5[26129] = {X 509.4595, Y 9.5048, Z -8.0000, A 0.000, B 0.000, C 0.000 }
gfCNCPoint5[26130] = {X 509.7408, Y 10.3715, Z -8.0000, A 0.000, B 0.000, C 0.000 }
gfCNCPoint5[26131] = {X 509.9113, Y 11.2666, Z -8.0000, A 0.000, B 0.000, C 0.000 }
gfCNCPoint5[26132] = {X 509.9685, Y 12.1759, Z -8.0000, A 0.000, B 0.000, C 0.000 }
gfCNCPoint5[26133] = {X 509.9682, Y 13.0462, Z -8.0000, A 0.000, B 0.000, C 0.000 }
gfCNCPoint5[26134] = {X 509.8612, Y 14.2233, Z -8.0000, A 0.000, B 0.000, C 0.000 }
gfCNCPoint5[26135] = {X 509.5651, Y 15.3676, Z -8.0000, A 0.000, B 0.000, C 0.000 }
gfCNCPoint5[26136] = {X 509.0878, Y 16.4489, Z -8.0000, A 0.000, B 0.000, C 0.000 }
gfCNCPoint5[26137] = {X 508.4418, Y 17.4387, Z -8.0000, A 0.000, B 0.000, C 0.000 }
gfCNCPoint5[26138] = {X 508.4423, Y 39.7488, Z -8.0000, A 0.000, B 0.000, C 0.000 }
gfCNCPoint5[26139] = {X 509.0899, Y 40.7418, Z -8.0000, A 0.000, B 0.000, C 0.000 }
gfCNCPoint5[26140] = {X 509.5678, Y 41.8268, Z -8.0000, A 0.000, B 0.000, C 0.000 }
gfCNCPoint5[26141] = {X 509.8632, Y 42.9749, Z -8.0000, A 0.000, B 0.000, C 0.000 }
gfCNCPoint5[26142] = {X 509.9683, Y 44.1558, Z -8.0000, A 0.000, B 0.000, C 0.000 }
gfCNCPoint5[26143] = {X 509.9685, Y 45.0000, Z -8.0000, A 0.000, B 0.000, C 0.000 }
gfCNCPoint5[26144] = {X 509.8909, Y 46.0603, Z -8.0000, A 0.000, B 0.000, C 0.000 }
gfCNCPoint5[26145] = {X 509.6596, Y 47.0980, Z -8.0000, A 0.000, B 0.000, C 0.000 }
gfCNCPoint5[26146] = {X 509.2797, Y 48.0910, Z -8.0000, A 0.000, B 0.000, C 0.000 }
gfCNCPoint5[26147] = {X 508.7593, Y 49.0180, Z -8.0000, A 0.000, B 0.000, C 0.000 }
gfCNCPoint5[26148] = {X 508.0200, Y 49.9571, Z -8.0000, A 0.000, B 0.000, C 0.000 }
gfCNCPoint5[26149] = {X 507.1371, Y 50.7626, Z -8.0000, A 0.000, B 0.000, C 0.000 }
gfCNCPoint5[26150] = {X 506.1343, Y 51.4129, Z -8.0000, A 0.000, B 0.000, C 0.000 }
gfCNCPoint5[26151] = {X 505.0386, Y 51.8902, Z -8.0000, A 0.000, B 0.000, C 0.000 }
gfCNCPoint5[26152] = {X 503.8796, Y 52.1819, Z -8.0000, A 0.000, B 0.000, C 0.000 }
gfCNCPoint5[26153] = {X 502.6885, Y 52.2800, Z -8.0000, A 0.000, B 0.000, C 0.000 }
gfCNCPoint5[26154] = {X 496.2450, Y 52.2800, Z -8.0000, A 0.000, B 0.000, C 0.000 }
gfCNCPoint5[26155] = {X 495.0845, Y 52.1869, Z -8.0000, A 0.000, B 0.000, C 0.000 }
gfCNCPoint5[26156] = {X 493.9538, Y 51.9100, Z -8.0000, A 0.000, B 0.000, C 0.000 }
gfCNCPoint5[26157] = {X 492.8816, Y 51.4564, Z -8.0000, A 0.000, B 0.000, C 0.000 }
gfCNCPoint5[26158] = {X 491.8954, Y 50.8377, Z -8.0000, A 0.000, B 0.000, C 0.000 }
gfCNCPoint5[26159] = {X 491.0204, Y 50.0697, Z -8.0000, A 0.000, B 0.000, C 0.000 }
gfCNCPoint5[26160] = {X 490.2980, Y 49.1989, Z -8.0000, A 0.000, B 0.000, C 0.000 }
gfCNCPoint5[26161] = {X 489.7192, Y 48.2267, Z -8.0000, A 0.000, B 0.000, C 0.000 }
gfCNCPoint5[26162] = {X 489.2980, Y 47.1766, Z -8.0000, A 0.000, B 0.000, C 0.000 }
gfCNCPoint5[26163] = {X 488.8769, Y 48.2267, Z -8.0000, A 0.000, B 0.000, C 0.000 }
gfCNCPoint5[26164] = {X 488.2981, Y 49.1989, Z -8.0000, A 0.000, B 0.000, C 0.000 }
gfCNCPoint5[26165] = {X 487.5756, Y 50.0697, Z -8.0000, A 0.000, B 0.000, C 0.000 }
gfCNCPoint5[26166] = {X 486.8824, Y 50.6978, Z -8.0000, A 0.000, B 0.000, C 0.000 }
gfCNCPoint5[26167] = {X 486.1145, Y 51.2318, Z -8.0000, A 0.000, B 0.000, C 0.000 }
gfCNCPoint5[26168] = {X 485.2843, Y 51.6629, Z -8.0000, A 0.000, B 0.000, C 0.000 }
gfCNCPoint5[26169] = {X 486.0586, Y 53.1385, Z -8.0000, A 0.000, B 0.000, C 0.000 }
gfCNCPoint5[26170] = {X 486.6224, Y 54.7067, Z -8.0000, A 0.000, B 0.000, C 0.000 }
gfCNCPoint5[26171] = {X 486.9651, Y 56.3375, Z -8.0000, A 0.000, B 0.000, C 0.000 }
gfCNCPoint5[26172] = {X 487.0800, Y 58.0000, Z -8.0000, A 0.000, B 0.000, C 0.000 }
gfCNCPoint5[26173] = {X 487.0796, Y 59.0339, Z -8.0000, A 0.000, B 0.000, C 0.000 }
gfCNCPoint5[26174] = {X 486.9597, Y 60.6349, Z -8.0000, A 0.000, B 0.000, C 0.000 }
gfCNCPoint5[26175] = {X 486.6285, Y 62.2060, Z -8.0000, A 0.000, B 0.000, C 0.000 }
gfCNCPoint5[26176] = {X 486.0918, Y 63.7192, Z -8.0000, A 0.000, B 0.000, C 0.000 }
gfCNCPoint5[26177] = {X 485.3593, Y 65.1479, Z -8.0000, A 0.000, B 0.000, C 0.000 }
gfCNCPoint5[26178] = {X 484.4437, Y 66.4669, Z -8.0000, A 0.000, B 0.000, C 0.000 }
gfCNCPoint5[26179] = {X 483.3613, Y 67.6527, Z -8.0000, A 0.000, B 0.000, C 0.000 }
gfCNCPoint5[26180] = {X 483.3616, Y 88.3516, Z -8.0000, A 0.000, B 0.000, C 0.000 }
gfCNCPoint5[26181] = {X 484.3108, Y 89.3720, Z -8.0000, A 0.000, B 0.000, C 0.000 }
gfCNCPoint5[26182] = {X 485.1359, Y 90.4952, Z -8.0000, A 0.000, B 0.000, C 0.000 }
gfCNCPoint5[26183] = {X 507.6811, Y 90.4952, Z -8.0000, A 0.000, B 0.000, C 0.000 }
gfCNCPoint5[26184] = {X 507.6811, Y 92.8952, Z -8.0000, A 0.000, B 0.000, C 0.000 }
gfCNCPoint5[26185] = {X 592.8967, Y 92.8952, Z -8.0000, A 0.000, B 0.000, C 0.000 }
gfCNCPoint5[26186] = {X 592.8967, Y 56.5812, Z -8.0000, A 0.000, B 0.000, C 0.000 }
gfCNCPoint5[26187] = {X 591.4811, Y 56.4128, Z -8.0000, A 0.000, B 0.000, C 0.000 }
gfCNCPoint5[26188] = {X 590.0968, Y 56.0721, Z -8.0000, A 0.000, B 0.000, C 0.000 }
gfCNCPoint5[26189] = {X 588.7648, Y 55.5641, Z -8.0000, A 0.000, B 0.000, C 0.000 }
gfCNCPoint5[26190] = {X 587.5052, Y 54.8965, Z -8.0000, A 0.000, B 0.000, C 0.000 }
gfCNCPoint5[26191] = {X 586.9690, Y 55.2051, Z -8.0000, A 0.000, B 0.000, C 0.000 }
gfCNCPoint5[26192] = {X 586.4171, Y 55.4846, Z -8.0000, A 0.000, B 0.000, C 0.000 }
gfCNCPoint5[26193] = {X 584.8782, Y 56.0830, Z -8.0000, A 0.000, B 0.000, C 0.000 }
gfCNCPoint5[26194] = {X 583.2699, Y 56.4570, Z -8.0000, A 0.000, B 0.000, C 0.000 }
gfCNCPoint5[26195] = {X 581.6248, Y 56.5987, Z -8.0000, A 0.000, B 0.000, C 0.000 }
gfCNCPoint5[26196] = {X 579.9763, Y 56.5055, Z -8.0000, A 0.000, B 0.000, C 0.000 }
gfCNCPoint5[26197] = {X 578.3577, Y 56.1792, Z -8.0000, A 0.000, B 0.000, C 0.000 }
gfCNCPoint5[26198] = {X 576.8018, Y 55.6263, Z -8.0000, A 0.000, B 0.000, C 0.000 }
gfCNCPoint5[26199] = {X 575.3401, Y 54.8581, Z -8.0000, A 0.000, B 0.000, C 0.000 }
gfCNCPoint5[26200] = {X 573.9176, Y 55.6091, Z -8.0000, A 0.000, B 0.000, C 0.000 }
gfCNCPoint5[26201] = {X 572.4049, Y 56.1560, Z -8.0000, A 0.000, B 0.000, C 0.000 }
gfCNCPoint5[26202] = {X 570.8311, Y 56.4885, Z -8.0000, A 0.000, B 0.000, C 0.000 }
gfCNCPoint5[26203] = {X 569.2264, Y 56.6000, Z -8.0000, A 0.000, B 0.000, C 0.000 }
gfCNCPoint5[26204] = {X 562.4443, Y 56.6000, Z -8.0000, A 0.000, B 0.000, C 0.000 }
gfCNCPoint5[26205] = {X 560.8794, Y 56.4940, Z -8.0000, A 0.000, B 0.000, C 0.000 }
gfCNCPoint5[26206] = {X 559.3430, Y 56.1778, Z -8.0000, A 0.000, B 0.000, C 0.000 }
gfCNCPoint5[26207] = {X 557.8634, Y 55.6572, Z -8.0000, A 0.000, B 0.000, C 0.000 }
gfCNCPoint5[26208] = {X 556.4676, Y 54.9418, Z -8.0000, A 0.000, B 0.000, C 0.000 }
gfCNCPoint5[26209] = {X 555.1810, Y 54.0446, Z -8.0000, A 0.000, B 0.000, C 0.000 }
gfCNCPoint5[26210] = {X 554.0272, Y 52.9820, Z -8.0000, A 0.000, B 0.000, C 0.000 }
gfCNCPoint5[26211] = {X 553.0273, Y 51.7735, Z -8.0000, A 0.000, B 0.000, C 0.000 }
gfCNCPoint5[26212] = {X 552.1996, Y 50.4411, Z -8.0000, A 0.000, B 0.000, C 0.000 }
gfCNCPoint5[26213] = {X 551.5592, Y 49.0093, Z -8.0000, A 0.000, B 0.000, C 0.000 }
gfCNCPoint5[26214] = {X 551.1639, Y 47.7040, Z -8.0000, A 0.000, B 0.000, C 0.000 }
gfCNCPoint5[26215] = {X 550.9245, Y 46.3614, Z -8.0000, A 0.000, B 0.000, C 0.000 }
gfCNCPoint5[26216] = {X 550.8443, Y 45.0000, Z -8.0000, A 0.000, B 0.000, C 0.000 }
gfCNCPoint5[26217] = {X 550.8443, Y 44.0420, Z -8.0000, A 0.000, B 0.000, C 0.000 }
gfCNCPoint5[26218] = {X 550.9578, Y 42.4576, Z -8.0000, A 0.000, B 0.000, C 0.000 }
gfCNCPoint5[26219] = {X 551.2862, Y 40.9034, Z -8.0000, A 0.000, B 0.000, C 0.000 }
gfCNCPoint5[26220] = {X 551.8233, Y 39.4085, Z -8.0000, A 0.000, B 0.000, C 0.000 }
gfCNCPoint5[26221] = {X 549.6253, Y 38.4446, Z -8.0000, A 0.000, B 0.000, C 0.000 }
gfCNCPoint5[26222] = {X 549.7927, Y 38.0773, Z -8.0000, A 0.000, B 0.000, C 0.000 }
gfCNCPoint5[26223] = {X 549.9706, Y 37.7150, Z -8.0000, A 0.000, B 0.000, C 0.000 }
gfCNCPoint5[26224] = {X 549.9709, Y 16.9523, Z -8.0000, A 0.000, B 0.000, C 0.000 }
gfCNCPoint5[26225] = {X 549.8033, Y 17.1984, Z -8.0000, A 0.000, B 0.000, C 0.000 }
gfCNCPoint5[26226] = {X 549.6258, Y 17.4374, Z -8.0000, A 0.000, B 0.000, C 0.000 }
gfCNCPoint5[26227] = {X 549.6253, Y 38.4446, Z -8.0000, A 0.000, B 0.000, C 0.000 }
gfCNCPoint5[26228] = {X 551.8233, Y 39.4085, Z -8.0000, A 0.000, B 0.000, C 0.000 }
gfCNCPoint5[26229] = {X 552.0827, Y 38.8568, Z -8.0000, A 0.000, B 0.000, C 0.000 }
gfCNCPoint5[26230] = {X 552.3706, Y 38.3194, Z -8.0000, A 0.000, B 0.000, C 0.000 }
gfCNCPoint5[26231] = {X 552.3710, Y 11.6863, Z -8.0000, A 0.000, B 0.000, C 0.000 }
gfCNCPoint5[26232] = {X 551.6701, Y 10.2324, Z -8.0000, A 0.000, B 0.000, C 0.000 }
gfCNCPoint5[26233] = {X 551.1777, Y 8.6954, Z -8.0000, A 0.000, B 0.000, C 0.000 }
gfCNCPoint5[26234] = {X 550.9035, Y 7.1048, Z -8.0000, A 0.000, B 0.000, C 0.000 }
gfCNCPoint5[26235] = {X 524.2926, Y 7.1048, Z -8.0000, A 0.000, B 0.000, C 0.000 }
gfCNCPoint5[26236] = {X 524.3782, Y 7.2059, Z -8.0000, A 0.000, B 0.000, C 0.000 }
gfCNCPoint5[26237] = {X 524.4609, Y 7.3092, Z -8.0000, A 0.000, B 0.000, C 0.000 }
gfCNCPoint5[26238] = {X 543.7426, Y 7.3092, Z -8.0000, A 0.000, B 0.000, C 0.000 }
gfCNCPoint5[26239] = {X 544.7121, Y 7.3813, Z -8.0000, A 0.000, B 0.000, C 0.000 }
gfCNCPoint5[26240] = {X 545.6481, Y 7.6440, Z -8.0000, A 0.000, B 0.000, C 0.000 }
gfCNCPoint5[26241] = {X 546.5136, Y 8.0869, Z -8.0000, A 0.000, B 0.000, C 0.000 }
gfCNCPoint5[26242] = {X 547.2742, Y 8.6924, Z -8.0000, A 0.000, B 0.000, C 0.000 }
gfCNCPoint5[26243] = {X 547.8998, Y 9.4365, Z -8.0000, A 0.000, B 0.000, C 0.000 }
gfCNCPoint5[26244] = {X 548.3657, Y 10.2898, Z -8.0000, A 0.000, B 0.000, C 0.000 }
gfCNCPoint5[26245] = {X 548.6534, Y 11.2184, Z -8.0000, A 0.000, B 0.000, C 0.000 }
gfCNCPoint5[26246] = {X 548.7514, Y 12.1856, Z -8.0000, A 0.000, B 0.000, C 0.000 }
gfCNCPoint5[26247] = {X 548.7512, Y 13.0237, Z -8.0000, A 0.000, B 0.000, C 0.000 }
gfCNCPoint5[26248] = {X 548.6554, Y 13.9415, Z -8.0000, A 0.000, B 0.000, C 0.000 }
gfCNCPoint5[26249] = {X 548.3885, Y 14.8248, Z -8.0000, A 0.000, B 0.000, C 0.000 }
gfCNCPoint5[26250] = {X 547.9601, Y 15.6421, Z -8.0000, A 0.000, B 0.000, C 0.000 }
gfCNCPoint5[26251] = {X 547.6189, Y 16.1039, Z -8.0000, A 0.000, B 0.000, C 0.000 }
gfCNCPoint5[26252] = {X 547.2258, Y 16.5224, Z -8.0000, A 0.000, B 0.000, C 0.000 }
gfCNCPoint5[26253] = {X 547.2253, Y 40.6639, Z -8.0000, A 0.000, B 0.000, C 0.000 }
gfCNCPoint5[26254] = {X 547.8661, Y 41.4057, Z -8.0000, A 0.000, B 0.000, C 0.000 }
gfCNCPoint5[26255] = {X 548.3457, Y 42.2607, Z -8.0000, A 0.000, B 0.000, C 0.000 }
gfCNCPoint5[26256] = {X 548.6448, Y 43.1942, Z -8.0000, A 0.000, B 0.000, C 0.000 }
gfCNCPoint5[26257] = {X 548.7513, Y 44.1687, Z -8.0000, A 0.000, B 0.000, C 0.000 }
gfCNCPoint5[26258] = {X 548.7514, Y 45.0006, Z -8.0000, A 0.000, B 0.000, C 0.000 }
gfCNCPoint5[26259] = {X 548.6700, Y 45.8824, Z -8.0000, A 0.000, B 0.000, C 0.000 }
gfCNCPoint5[26260] = {X 548.4307, Y 46.7351, Z -8.0000, A 0.000, B 0.000, C 0.000 }
gfCNCPoint5[26261] = {X 548.0413, Y 47.5306, Z -8.0000, A 0.000, B 0.000, C 0.000 }
gfCNCPoint5[26262] = {X 547.5147, Y 48.2427, Z -8.0000, A 0.000, B 0.000, C 0.000 }
gfCNCPoint5[26263] = {X 546.7291, Y 48.9524, Z -8.0000, A 0.000, B 0.000, C 0.000 }
gfCNCPoint5[26264] = {X 545.8090, Y 49.4762, Z -8.0000, A 0.000, B 0.000, C 0.000 }
gfCNCPoint5[26265] = {X 544.7977, Y 49.7893, Z -8.0000, A 0.000, B 0.000, C 0.000 }
gfCNCPoint5[26266] = {X 543.7426, Y 49.8773, Z -8.0000, A 0.000, B 0.000, C 0.000 }
gfCNCPoint5[26267] = {X 524.3241, Y 49.8776, Z -8.0000, A 0.000, B 0.000, C 0.000 }
gfCNCPoint5[26268] = {X 523.7111, Y 50.5164, Z -8.0000, A 0.000, B 0.000, C 0.000 }
gfCNCPoint5[26269] = {X 522.9958, Y 51.0379, Z -8.0000, A 0.000, B 0.000, C 0.000 }
gfCNCPoint5[26270] = {X 522.2002, Y 51.4262, Z -8.0000, A 0.000, B 0.000, C 0.000 }
gfCNCPoint5[26271] = {X 521.3489, Y 51.6691, Z -8.0000, A 0.000, B 0.000, C 0.000 }
gfCNCPoint5[26272] = {X 520.4681, Y 51.7591, Z -8.0000, A 0.000, B 0.000, C 0.000 }
gfCNCPoint5[26273] = {X 519.7998, Y 51.7591, Z -8.0000, A 0.000, B 0.000, C 0.000 }
gfCNCPoint5[26274] = {X 518.8477, Y 51.6654, Z -8.0000, A 0.000, B 0.000, C 0.000 }
gfCNCPoint5[26275] = {X 517.9323, Y 51.3877, Z -8.0000, A 0.000, B 0.000, C 0.000 }
gfCNCPoint5[26276] = {X 517.0886, Y 50.9367, Z -8.0000, A 0.000, B 0.000, C 0.000 }
gfCNCPoint5[26277] = {X 516.3491, Y 50.3298, Z -8.0000, A 0.000, B 0.000, C 0.000 }
gfCNCPoint5[26278] = {X 515.7422, Y 49.5903, Z -8.0000, A 0.000, B 0.000, C 0.000 }
gfCNCPoint5[26279] = {X 515.2912, Y 48.7466, Z -8.0000, A 0.000, B 0.000, C 0.000 }
gfCNCPoint5[26280] = {X 515.0135, Y 47.8312, Z -8.0000, A 0.000, B 0.000, C 0.000 }
gfCNCPoint5[26281] = {X 514.9198, Y 46.8791, Z -8.0000, A 0.000, B 0.000, C 0.000 }
gfCNCPoint5[26282] = {X 514.9198, Y 39.9011, Z -8.0000, A 0.000, B 0.000, C 0.000 }
gfCNCPoint5[26283] = {X 515.0197, Y 38.9186, Z -8.0000, A 0.000, B 0.000, C 0.000 }
gfCNCPoint5[26284] = {X 515.3154, Y 37.9764, Z -8.0000, A 0.000, B 0.000, C 0.000 }
gfCNCPoint5[26285] = {X 515.7947, Y 37.1129, Z -8.0000, A 0.000, B 0.000, C 0.000 }
gfCNCPoint5[26286] = {X 516.4381, Y 36.3637, Z -8.0000, A 0.000, B 0.000, C 0.000 }
gfCNCPoint5[26287] = {X 517.2191, Y 35.7593, Z -8.0000, A 0.000, B 0.000, C 0.000 }
gfCNCPoint5[26288] = {X 518.1058, Y 35.3245, Z -8.0000, A 0.000, B 0.000, C 0.000 }
gfCNCPoint5[26289] = {X 519.0619, Y 35.0772, Z -8.0000, A 0.000, B 0.000, C 0.000 }
gfCNCPoint5[26290] = {X 519.4084, Y 35.0368, Z -8.0000, A 0.000, B 0.000, C 0.000 }
gfCNCPoint5[26291] = {X 519.7568, Y 35.0213, Z -8.0000, A 0.000, B 0.000, C 0.000 }
gfCNCPoint5[26292] = {X 520.5345, Y 35.0216, Z -8.0000, A 0.000, B 0.000, C 0.000 }
gfCNCPoint5[26293] = {X 521.4082, Y 35.1125, Z -8.0000, A 0.000, B 0.000, C 0.000 }
gfCNCPoint5[26294] = {X 522.2515, Y 35.3586, Z -8.0000, A 0.000, B 0.000, C 0.000 }
gfCNCPoint5[26295] = {X 523.0370, Y 35.7519, Z -8.0000, A 0.000, B 0.000, C 0.000 }
gfCNCPoint5[26296] = {X 523.7392, Y 36.2797, Z -8.0000, A 0.000, B 0.000, C 0.000 }
gfCNCPoint5[26297] = {X 524.3355, Y 36.9248, Z -8.0000, A 0.000, B 0.000, C 0.000 }
gfCNCPoint5[26298] = {X 534.0719, Y 36.9248, Z -8.0000, A 0.000, B 0.000, C 0.000 }
gfCNCPoint5[26299] = {X 534.0719, Y 34.5264, Z -8.0000, A 0.000, B 0.000, C 0.000 }
gfCNCPoint5[26300] = {X 530.3953, Y 34.5263, Z -8.0000, A 0.000, B 0.000, C 0.000 }
gfCNCPoint5[26301] = {X 529.7954, Y 35.1745, Z -8.0000, A 0.000, B 0.000, C 0.000 }
gfCNCPoint5[26302] = {X 529.0886, Y 35.7040, Z -8.0000, A 0.000, B 0.000, C 0.000 }
gfCNCPoint5[26303] = {X 528.2978, Y 36.0974, Z -8.0000, A 0.000, B 0.000, C 0.000 }
gfCNCPoint5[26304] = {X 527.4491, Y 36.3418, Z -8.0000, A 0.000, B 0.000, C 0.000 }
gfCNCPoint5[26305] = {X 526.5703, Y 36.4293, Z -8.0000, A 0.000, B 0.000, C 0.000 }
gfCNCPoint5[26306] = {X 525.8868, Y 36.4294, Z -8.0000, A 0.000, B 0.000, C 0.000 }
gfCNCPoint5[26307] = {X 524.9094, Y 36.3306, Z -8.0000, A 0.000, B 0.000, C 0.000 }
gfCNCPoint5[26308] = {X 523.9717, Y 36.0380, Z -8.0000, A 0.000, B 0.000, C 0.000 }
gfCNCPoint5[26309] = {X 523.1116, Y 35.5636, Z -8.0000, A 0.000, B 0.000, C 0.000 }
gfCNCPoint5[26310] = {X 522.3639, Y 34.9265, Z -8.0000, A 0.000, B 0.000, C 0.000 }
gfCNCPoint5[26311] = {X 521.7590, Y 34.1525, Z -8.0000, A 0.000, B 0.000, C 0.000 }
gfCNCPoint5[26312] = {X 521.3213, Y 33.2731, Z -8.0000, A 0.000, B 0.000, C 0.000 }
gfCNCPoint5[26313] = {X 521.0686, Y 32.3239, Z -8.0000, A 0.000, B 0.000, C 0.000 }
gfCNCPoint5[26314] = {X 521.0222, Y 31.9379, Z -8.0000, A 0.000, B 0.000, C 0.000 }
gfCNCPoint5[26315] = {X 521.0068, Y 31.5495, Z -8.0000, A 0.000, B 0.000, C 0.000 }
gfCNCPoint5[26316] = {X 521.0076, Y 24.4815, Z -8.0000, A 0.000, B 0.000, C 0.000 }
gfCNCPoint5[26317] = {X 521.0984, Y 23.6300, Z -8.0000, A 0.000, B 0.000, C 0.000 }
gfCNCPoint5[26318] = {X 521.3368, Y 22.8074, Z -8.0000, A 0.000, B 0.000, C 0.000 }
gfCNCPoint5[26319] = {X 521.7152, Y 22.0391, Z -8.0000, A 0.000, B 0.000, C 0.000 }
gfCNCPoint5[26320] = {X 521.1864, Y 22.1316, Z -8.0000, A 0.000, B 0.000, C 0.000 }
gfCNCPoint5[26321] = {X 520.6505, Y 22.1656, Z -8.0000, A 0.000, B 0.000, C 0.000 }
gfCNCPoint5[26322] = {X 519.9691, Y 22.1657, Z -8.0000, A 0.000, B 0.000, C 0.000 }
gfCNCPoint5[26323] = {X 519.5109, Y 22.1442, Z -8.0000, A 0.000, B 0.000, C 0.000 }
gfCNCPoint5[26324] = {X 519.0567, Y 22.0797, Z -8.0000, A 0.000, B 0.000, C 0.000 }
gfCNCPoint5[26325] = {X 518.1336, Y 21.8074, Z -8.0000, A 0.000, B 0.000, C 0.000 }
gfCNCPoint5[26326] = {X 517.2820, Y 21.3592, Z -8.0000, A 0.000, B 0.000, C 0.000 }
gfCNCPoint5[26327] = {X 516.5348, Y 20.7527, Z -8.0000, A 0.000, B 0.000, C 0.000 }
gfCNCPoint5[26328] = {X 515.9212, Y 20.0113, Z -8.0000, A 0.000, B 0.000, C 0.000 }
gfCNCPoint5[26329] = {X 515.4650, Y 19.1639, Z -8.0000, A 0.000, B 0.000, C 0.000 }
gfCNCPoint5[26330] = {X 515.1840, Y 18.2434, Z -8.0000, A 0.000, B 0.000, C 0.000 }
gfCNCPoint5[26331] = {X 515.0891, Y 17.2857, Z -8.0000, A 0.000, B 0.000, C 0.000 }
gfCNCPoint5[26332] = {X 515.0891, Y 10.3077, Z -8.0000, A 0.000, B 0.000, C 0.000 }
gfCNCPoint5[26333] = {X 515.0966, Y 10.0382, Z -8.0000, A 0.000, B 0.000, C 0.000 }
gfCNCPoint5[26334] = {X 515.1189, Y 9.7695, Z -8.0000, A 0.000, B 0.000, C 0.000 }
gfCNCPoint5[26335] = {X 515.3252, Y 8.8082, Z -8.0000, A 0.000, B 0.000, C 0.000 }
gfCNCPoint5[26336] = {X 515.7200, Y 7.9078, Z -8.0000, A 0.000, B 0.000, C 0.000 }
gfCNCPoint5[26337] = {X 516.2873, Y 7.1048, Z -8.0000, A 0.000, B 0.000, C 0.000 }
gfCNCPoint5[26338] = {X 516.6494, Y 7.4199, Z -8.0000, A 0.000, B 0.000, C 0.000 }
gfCNCPoint5[26339] = {X 517.3374, Y 6.7815, Z -8.0000, A 0.000, B 0.000, C 0.000 }
gfCNCPoint5[26340] = {X 518.1452, Y 6.3035, Z -8.0000, A 0.000, B 0.000, C 0.000 }
gfCNCPoint5[26341] = {X 519.0360, Y 6.0078, Z -8.0000, A 0.000, B 0.000, C 0.000 }
gfCNCPoint5[26342] = {X 519.9692, Y 5.9077, Z -8.0000, A 0.000, B 0.000, C 0.000 }
gfCNCPoint5[26343] = {X 520.6509, Y 5.9079, Z -8.0000, A 0.000, B 0.000, C 0.000 }
gfCNCPoint5[26344] = {X 521.4831, Y 5.9950, Z -8.0000, A 0.000, B 0.000, C 0.000 }
gfCNCPoint5[26345] = {X 522.2837, Y 6.2381, Z -8.0000, A 0.000, B 0.000, C 0.000 }
gfCNCPoint5[26346] = {X 523.0239, Y 6.6284, Z -8.0000, A 0.000, B 0.000, C 0.000 }
gfCNCPoint5[26347] = {X 523.6767, Y 7.1518, Z -8.0000, A 0.000, B 0.000, C 0.000 }
gfCNCPoint5[26348] = {X 524.2187, Y 7.7892, Z -8.0000, A 0.000, B 0.000, C 0.000 }
gfCNCPoint5[26349] = {X 543.7489, Y 7.7892, Z -8.0000, A 0.000, B 0.000, C 0.000 }
gfCNCPoint5[26350] = {X 544.7473, Y 7.8766, Z -8.0000, A 0.000, B 0.000, C 0.000 }
gfCNCPoint5[26351] = {X 545.7001, Y 8.1873, Z -8.0000, A 0.000, B 0.000, C 0.000 }
gfCNCPoint5[26352] = {X 546.5580, Y 8.7054, Z -8.0000, A 0.000, B 0.000, C 0.000 }
gfCNCPoint5[26353] = {X 547.2766, Y 9.4040, Z -8.0000, A 0.000, B 0.000, C 0.000 }
gfCNCPoint5[26354] = {X 547.8186, Y 10.2470, Z -8.0000, A 0.000, B 0.000, C 0.000 }
gfCNCPoint5[26355] = {X 548.1561, Y 11.1907, Z -8.0000, A 0.000, B 0.000, C 0.000 }
gfCNCPoint5[26356] = {X 548.2714, Y 12.1863, Z -8.0000, A 0.000, B 0.000, C 0.000 }
gfCNCPoint5[26357] = {X 548.2712, Y 13.0233, Z -8.0000, A 0.000, B 0.000, C 0.000 }
gfCNCPoint5[26358] = {X 548.1630, Y 13.9487, Z -8.0000, A 0.000, B 0.000, C 0.000 }
gfCNCPoint5[26359] = {X 547.8624, Y 14.8306, Z -8.0000, A 0.000, B 0.000, C 0.000 }
gfCNCPoint5[26360] = {X 547.3828, Y 15.6295, Z -8.0000, A 0.000, B 0.000, C 0.000 }
gfCNCPoint5[26361] = {X 546.7458, Y 16.3094, Z -8.0000, A 0.000, B 0.000, C 0.000 }
gfCNCPoint5[26362] = {X 546.7453, Y 40.8770, Z -8.0000, A 0.000, B 0.000, C 0.000 }
gfCNCPoint5[26363] = {X 547.3893, Y 41.5660, Z -8.0000, A 0.000, B 0.000, C 0.000 }
gfCNCPoint5[26364] = {X 547.8717, Y 42.3765, Z -8.0000, A 0.000, B 0.000, C 0.000 }
gfCNCPoint5[26365] = {X 548.1704, Y 43.2711, Z -8.0000, A 0.000, B 0.000, C 0.000 }
gfCNCPoint5[26366] = {X 548.2714, Y 44.2089, Z -8.0000, A 0.000, B 0.000, C 0.000 }
gfCNCPoint5[26367] = {X 548.2714, Y 45.0006, Z -8.0000, A 0.000, B 0.000, C 0.000 }
gfCNCPoint5[26368] = {X 548.1560, Y 45.9961, Z -8.0000, A 0.000, B 0.000, C 0.000 }
gfCNCPoint5[26369] = {X 547.8185, Y 46.9397, Z -8.0000, A 0.000, B 0.000, C 0.000 }
gfCNCPoint5[26370] = {X 547.2765, Y 47.7826, Z -8.0000, A 0.000, B 0.000, C 0.000 }
gfCNCPoint5[26371] = {X 546.5579, Y 48.4812, Z -8.0000, A 0.000, B 0.000, C 0.000 }
gfCNCPoint5[26372] = {X 545.7000, Y 48.9993, Z -8.0000, A 0.000, B 0.000, C 0.000 }
gfCNCPoint5[26373] = {X 544.7472, Y 49.3100, Z -8.0000, A 0.000, B 0.000, C 0.000 }
gfCNCPoint5[26374] = {X 543.7489, Y 49.3973, Z -8.0000, A 0.000, B 0.000, C 0.000 }
gfCNCPoint5[26375] = {X 524.0868, Y 49.3976, Z -8.0000, A 0.000, B 0.000, C 0.000 }
gfCNCPoint5[26376] = {X 523.5299, Y 50.0325, Z -8.0000, A 0.000, B 0.000, C 0.000 }
gfCNCPoint5[26377] = {X 522.8654, Y 50.5537, Z -8.0000, A 0.000, B 0.000, C 0.000 }
gfCNCPoint5[26378] = {X 522.1161, Y 50.9433, Z -8.0000, A 0.000, B 0.000, C 0.000 }
gfCNCPoint5[26379] = {X 521.3078, Y 51.1879, Z -8.0000, A 0.000, B 0.000, C 0.000 }
